LIN {X 0,Y 568.103,Z 672.069,A -85,B 0,C 180,E1 27364.138,E2 27364.138} C_VEL
LIN {X 0,Y 568.021,Z 680.785,A -85,B 0,C 180,E1 27362.825,E2 27362.825} C_VEL
LIN {X 0,Y 567.96,Z 688.715,A -85,B 0,C 180,E1 27361.312,E2 27361.312} C_VEL
LIN {X 0,Y 567.932,Z 694.6,A -85,B 0,C 180,E1 27359.799,E2 27359.799} C_VEL
LIN {X 0,Y 567.918,Z 698.81,A -85,B 0,C 180,E1 27358.285,E2 27358.285} C_VEL
LIN {X 0,Y 567.916,Z 701.625,A -85,B 0,C 180,E1 27356.569,E2 27356.569} C_VEL
LIN {X 0,Y 567.916,Z 702.444,A -85,B 0,C 180,E1 27355.051,E2 27355.051} C_VEL
LIN {X 0,Y 567.916,Z 701.73,A -85,B 0,C 180,E1 27353.429,E2 27353.429} C_VEL
LIN {X 0,Y 567.916,Z 698.96,A -85,B 0,C 180,E1 27351.7,E2 27351.7} C_VEL
LIN {X 0,Y 567.93,Z 694.8,A -85,B 0,C 180,E1 27350.168,E2 27350.168} C_VEL
LIN {X 0,Y 567.961,Z 688.386,A -85,B 0,C 180,E1 27348.526,E2 27348.526} C_VEL
LIN {X 0,Y 568.019,Z 680.765,A -85,B 0,C 180,E1 27347.083,E2 27347.083} C_VEL
LIN {X 0,Y 568.11,Z 671.85,A -85,B 0,C 180,E1 27345.736,E2 27345.736} C_VEL
LIN {X 0,Y 568.235,Z 660.961,A -85,B 0,C 180,E1 27344.435,E2 27344.435} C_VEL
LIN {X 0,Y 568.372,Z 650.225,A -85,B 0,C 180,E1 27343.39,E2 27343.39} C_VEL
LIN {X 0,Y 568.548,Z 637.033,A -85,B 0,C 180,E1 27342.341,E2 27342.341} C_VEL
LIN {X 0,Y 568.727,Z 623.6,A -85,B 0,C 180,E1 27341.502,E2 27341.502} C_VEL
LIN {X 0,Y 568.875,Z 610.751,A -85,B 0,C 180,E1 27340.865,E2 27340.865} C_VEL
LIN {X 0,Y 569.043,Z 595.744,A -85,B 0,C 180,E1 27340.299,E2 27340.299} C_VEL
LIN {X 0,Y 569.158,Z 579.316,A -85,B 0,C 180,E1 27339.884,E2 27339.884} C_VEL
LIN {X 0,Y 569.352,Z 502.923,A -85,B 0,C 180,E1 27338.879,E2 27338.879} C_VEL
LIN {X 0,Y 569.278,Z 438.341,A -85,B 0,C 180,E1 27338.045,E2 27338.045} C_VEL
LIN {X 0,Y 568.987,Z 435.852,A -85,B 0,C 180,E1 27337.992,E2 27337.992} C_VEL
LIN {X 0,Y 569.451,Z 392.592,A -85,B 0,C 180,E1 27334.633,E2 27334.633} C_VEL
LIN {X 0,Y 569.848,Z 350.919,A -85,B 0,C 180,E1 27331.38,E2 27331.38} C_VEL
LIN {X 0,Y 569.783,Z 320.283,A -85,B 0,C 180,E1 27329.105,E2 27329.105} C_VEL
LIN {X 0,Y 569.208,Z 278.696,A -85,B 0,C 180,E1 27326.163,E2 27326.163} C_VEL
LIN {X 0,Y 568.41,Z 243.021,A -85,B 0,C 180,E1 27323.843,E2 27323.843} C_VEL
LIN {X 0,Y 568.206,Z 241.959,A -85,B 0,C 180,E1 27323.755,E2 27323.755} C_VEL
LIN {X 0,Y 568.249,Z 242.205,A -85,B 0,C 180,E1 27322.262,E2 27322.262} C_VEL
LIN {X 0,Y 569.363,Z 245.218,A -85,B 0,C 180,E1 27321.947,E2 27321.947} C_VEL
LIN {X 0,Y 575.363,Z 257.407,A -85,B 0,C 180,E1 27320.568,E2 27320.568} C_VEL
LIN {X 0,Y 574.722,Z 312.789,A -85,B 0,C 180,E1 27316.944,E2 27316.944} C_VEL
LIN {X 0,Y 576.412,Z 325.558,A -85,B 0,C 180,E1 27315.996,E2 27315.996} C_VEL
LIN {X 0,Y 579.316,Z 335.026,A -85,B 0,C 180,E1 27315.183,E2 27315.183} C_VEL
LIN {X 0,Y 583.109,Z 341.733,A -85,B 0,C 180,E1 27314.495,E2 27314.495} C_VEL
LIN {X 0,Y 587.828,Z 346.751,A -85,B 0,C 180,E1 27313.847,E2 27313.847} C_VEL
LIN {X 0,Y 591.052,Z 348.878,A -85,B 0,C 180,E1 27313.33,E2 27313.33} C_VEL
LIN {X 0,Y 593.631,Z 349.586,A -85,B 0,C 180,E1 27312.747,E2 27312.747} C_VEL
LIN {X 0,Y 595.105,Z 348.922,A -85,B 0,C 180,E1 27312.189,E2 27312.189} C_VEL
LIN {X 0,Y 595.528,Z 346.951,A -85,B 0,C 180,E1 27311.608,E2 27311.608} C_VEL
LIN {X 0,Y 594.698,Z 343.734,A -85,B 0,C 180,E1 27311.069,E2 27311.069} C_VEL
LIN {X 0,Y 592.583,Z 339.307,A -85,B 0,C 180,E1 27310.608,E2 27310.608} C_VEL
LIN {X 0,Y 588.547,Z 331.567,A -85,B 0,C 180,E1 27310.129,E2 27310.129} C_VEL
LIN {X 0,Y 585.378,Z 322.433,A -85,B 0,C 180,E1 27309.759,E2 27309.759} C_VEL
LIN {X 0,Y 583.166,Z 311.682,A -85,B 0,C 180,E1 27309.497,E2 27309.497} C_VEL
LIN {X 0,Y 581.969,Z 298.964,A -85,B 0,C 180,E1 27309.355,E2 27309.355} C_VEL
LIN {X 0,Y 581.754,Z 282.03,A -85,B 0,C 180,E1 27309.329,E2 27309.329} C_VEL
LIN {X 0,Y 581.598,Z 258.822,A -85,B 0,C 180,E1 27309.31,E2 27309.31} C_VEL
LIN {X 0,Y 577.973,Z 254.412,A -85,B 0,C 180,E1 27308.869,E2 27308.869} C_VEL
LIN {X 0,Y 574.072,Z 250.389,A -85,B 0,C 180,E1 27308.383,E2 27308.383} C_VEL
LIN {X 0,Y 571.751,Z 250.051,A -85,B 0,C 180,E1 27308.089,E2 27308.089} C_VEL
LIN {X 0,Y 571.629,Z 250.115,A -85,B 0,C 180,E1 27308.043,E2 27308.043} C_VEL
LIN {X 0,Y 573.988,Z 255.905,A -85,B 0,C 180,E1 27307.482,E2 27307.482} C_VEL
LIN {X 0,Y 573.245,Z 302.662,A -85,B 0,C 180,E1 27304.587,E2 27304.587} C_VEL
LIN {X 0,Y 574.384,Z 310.581,A -85,B 0,C 180,E1 27304.391,E2 27304.391} C_VEL
LIN {X 0,Y 573.271,Z 530.669,A -85,B 0,C 180,E1 27301.252,E2 27301.252} C_VEL
LIN {X 0,Y 572.868,Z 608.931,A -85,B 0,C 180,E1 27300.126,E2 27300.126} C_VEL
LIN {X 0,Y 572.55,Z 630.865,A -85,B 0,C 180,E1 27299.618,E2 27299.618} C_VEL
LIN {X 0,Y 572.128,Z 653.445,A -85,B 0,C 180,E1 27298.89,E2 27298.89} C_VEL
LIN {X 0,Y 571.709,Z 674.688,A -85,B 0,C 180,E1 27298.001,E2 27298.001} C_VEL
LIN {X 0,Y 571.187,Z 694.756,A -85,B 0,C 180,E1 27296.961,E2 27296.961} C_VEL
LIN {X 0,Y 570.674,Z 714.156,A -85,B 0,C 180,E1 27295.754,E2 27295.754} C_VEL
LIN {X 0,Y 570.184,Z 732.799,A -85,B 0,C 180,E1 27294.391,E2 27294.391} C_VEL
LIN {X 0,Y 569.662,Z 751.692,A -85,B 0,C 180,E1 27292.769,E2 27292.769} C_VEL
LIN {X 0,Y 569.196,Z 769.23,A -85,B 0,C 180,E1 27290.999,E2 27290.999} C_VEL
LIN {X 0,Y 568.818,Z 784.581,A -85,B 0,C 180,E1 27289.19,E2 27289.19} C_VEL
LIN {X 0,Y 568.521,Z 798.676,A -85,B 0,C 180,E1 27287.259,E2 27287.259} C_VEL
LIN {X 0,Y 568.303,Z 810.938,A -85,B 0,C 180,E1 27285.302,E2 27285.302} C_VEL
LIN {X 0,Y 568.132,Z 821.9,A -85,B 0,C 180,E1 27283.226,E2 27283.226} C_VEL
LIN {X 0,Y 568.021,Z 830.897,A -85,B 0,C 180,E1 27281.165,E2 27281.165} C_VEL
LIN {X 0,Y 567.965,Z 838.562,A -85,B 0,C 180,E1 27279.014,E2 27279.014} C_VEL
LIN {X 0,Y 567.933,Z 844.578,A -85,B 0,C 180,E1 27276.817,E2 27276.817} C_VEL
LIN {X 0,Y 567.916,Z 848.793,A -85,B 0,C 180,E1 27274.645,E2 27274.645} C_VEL
LIN {X 0,Y 567.909,Z 851.489,A -85,B 0,C 180,E1 27272.422,E2 27272.422} C_VEL
LIN {X 0,Y 567.905,Z 852.475,A -85,B 0,C 180,E1 27270.202,E2 27270.202} C_VEL
LIN {X 0,Y 567.912,Z 851.758,A -85,B 0,C 180,E1 27267.982,E2 27267.982} C_VEL
LIN {X 0,Y 567.914,Z 849.426,A -85,B 0,C 180,E1 27265.759,E2 27265.759} C_VEL
LIN {X 0,Y 567.915,Z 845.586,A -85,B 0,C 180,E1 27263.632,E2 27263.632} C_VEL
LIN {X 0,Y 567.937,Z 840.08,A -85,B 0,C 180,E1 27261.496,E2 27261.496} C_VEL
LIN {X 0,Y 567.996,Z 833.316,A -85,B 0,C 180,E1 27259.451,E2 27259.451} C_VEL
LIN {X 0,Y 568.086,Z 824.764,A -85,B 0,C 180,E1 27257.394,E2 27257.394} C_VEL
LIN {X 0,Y 568.235,Z 813.833,A -85,B 0,C 180,E1 27255.218,E2 27255.218} C_VEL
LIN {X 0,Y 568.458,Z 801.998,A -85,B 0,C 180,E1 27253.234,E2 27253.234} C_VEL
LIN {X 0,Y 568.759,Z 787.904,A -85,B 0,C 180,E1 27251.234,E2 27251.234} C_VEL
LIN {X 0,Y 569.106,Z 773.042,A -85,B 0,C 180,E1 27249.428,E2 27249.428} C_VEL
LIN {X 0,Y 569.526,Z 756.535,A -85,B 0,C 180,E1 27247.698,E2 27247.698} C_VEL
LIN {X 0,Y 569.994,Z 738.779,A -85,B 0,C 180,E1 27246.095,E2 27246.095} C_VEL
LIN {X 0,Y 570.521,Z 720.526,A -85,B 0,C 180,E1 27244.683,E2 27244.683} C_VEL
LIN {X 0,Y 571.06,Z 700.433,A -85,B 0,C 180,E1 27243.37,E2 27243.37} C_VEL
LIN {X 0,Y 571.525,Z 680.177,A -85,B 0,C 180,E1 27242.266,E2 27242.266} C_VEL
LIN {X 0,Y 572.038,Z 659.333,A -85,B 0,C 180,E1 27241.335,E2 27241.335} C_VEL
LIN {X 0,Y 572.456,Z 637.558,A -85,B 0,C 180,E1 27240.574,E2 27240.574} C_VEL
LIN {X 0,Y 572.759,Z 615.949,A -85,B 0,C 180,E1 27240.017,E2 27240.017} C_VEL
LIN {X 0,Y 573.002,Z 591.483,A -85,B 0,C 180,E1 27239.601,E2 27239.601} C_VEL
LIN {X 0,Y 574.056,Z 367.034,A -85,B 0,C 180,E1 27236.421,E2 27236.421} C_VEL
LIN {X 0,Y 574.187,Z 309.846,A -85,B 0,C 180,E1 27235.584,E2 27235.584} C_VEL
LIN {X 0,Y 572.736,Z 302.398,A -85,B 0,C 180,E1 27235.347,E2 27235.347} C_VEL
LIN {X 0,Y 573.538,Z 262.173,A -85,B 0,C 180,E1 27232.398,E2 27232.398} C_VEL
LIN {X 0,Y 573.705,Z 255.551,A -85,B 0,C 180,E1 27231.905,E2 27231.905} C_VEL
LIN {X 0,Y 573.143,Z 254.07,A -85,B 0,C 180,E1 27231.734,E2 27231.734} C_VEL
LIN {X 0,Y 575.005,Z 254.784,A -85,B 0,C 180,E1 27231.5,E2 27231.5} C_VEL
LIN {X 0,Y 577.504,Z 253.868,A -85,B 0,C 180,E1 27231.189,E2 27231.189} C_VEL
LIN {X 0,Y 581.598,Z 258.84,A -85,B 0,C 180,E1 27230.69,E2 27230.69} C_VEL
LIN {X 0,Y 581.762,Z 267.678,A -85,B 0,C 180,E1 27230.67,E2 27230.67} C_VEL
LIN {X 0,Y 581.94,Z 336.852,A -85,B 0,C 180,E1 27230.649,E2 27230.649} C_VEL
LIN {X 0,Y 583.106,Z 349.267,A -85,B 0,C 180,E1 27230.51,E2 27230.51} C_VEL
LIN {X 0,Y 585.298,Z 359.813,A -85,B 0,C 180,E1 27230.25,E2 27230.25} C_VEL
LIN {X 0,Y 588.468,Z 368.899,A -85,B 0,C 180,E1 27229.88,E2 27229.88} C_VEL
LIN {X 0,Y 591.818,Z 375.728,A -85,B 0,C 180,E1 27229.456,E2 27229.456} C_VEL
LIN {X 0,Y 593.551,Z 380.22,A -85,B 0,C 180,E1 27228.985,E2 27228.985} C_VEL
LIN {X 0,Y 594.01,Z 383.359,A -85,B 0,C 180,E1 27228.456,E2 27228.456} C_VEL
LIN {X 0,Y 593.268,Z 385.325,A -85,B 0,C 180,E1 27227.863,E2 27227.863} C_VEL
LIN {X 0,Y 591.619,Z 385.905,A -85,B 0,C 180,E1 27227.321,E2 27227.321} C_VEL
LIN {X 0,Y 588.94,Z 385.128,A -85,B 0,C 180,E1 27226.746,E2 27226.746} C_VEL
LIN {X 0,Y 585.706,Z 382.882,A -85,B 0,C 180,E1 27226.228,E2 27226.228} C_VEL
LIN {X 0,Y 580.98,Z 377.491,A -85,B 0,C 180,E1 27225.537,E2 27225.537} C_VEL
LIN {X 0,Y 577.144,Z 369.886,A -85,B 0,C 180,E1 27224.741,E2 27224.741} C_VEL
LIN {X 0,Y 574.585,Z 359.77,A -85,B 0,C 180,E1 27223.834,E2 27223.834} C_VEL
LIN {X 0,Y 573.474,Z 347.302,A -85,B 0,C 180,E1 27222.841,E2 27222.841} C_VEL
LIN {X 0,Y 574.378,Z 298.185,A -85,B 0,C 180,E1 27219.19,E2 27219.19} C_VEL
LIN {X 0,Y 575.319,Z 262.814,A -85,B 0,C 180,E1 27216.422,E2 27216.422} C_VEL
LIN {X 0,Y 575.444,Z 257.912,A -85,B 0,C 180,E1 27216.026,E2 27216.026} C_VEL
LIN {X 0,Y 569.719,Z 245.758,A -85,B 0,C 180,E1 27214.41,E2 27214.41} C_VEL
LIN {X 0,Y 568.261,Z 242.304,A -85,B 0,C 180,E1 27213.952,E2 27213.952} C_VEL
LIN {X 0,Y 568.218,Z 241.96,A -85,B 0,C 180,E1 27213.844,E2 27213.844} C_VEL
LIN {X 0,Y 568.212,Z 241.956,A -85,B 0,C 180,E1 27210.566,E2 27210.566} C_VEL
LIN {X 0,Y 568.193,Z 241.957,A -85,B 0,C 180,E1 27207.294,E2 27207.294} C_VEL
LIN {X 0,Y 568.248,Z 242.138,A -85,B 0,C 180,E1 27206.772,E2 27206.772} C_VEL
LIN {X 0,Y 568.786,Z 246.032,A -85,B 0,C 180,E1 27206.519,E2 27206.519} C_VEL
LIN {X 0,Y 569.334,Z 290.314,A -85,B 0,C 180,E1 27203.713,E2 27203.713} C_VEL
LIN {X 0,Y 569.709,Z 330.255,A -85,B 0,C 180,E1 27201.027,E2 27201.027} C_VEL
LIN {X 0,Y 569.686,Z 369.499,A -85,B 0,C 180,E1 27198.283,E2 27198.283} C_VEL
LIN {X 0,Y 569.314,Z 415.814,A -85,B 0,C 180,E1 27194.961,E2 27194.961} C_VEL
LIN {X 0,Y 568.878,Z 462.441,A -85,B 0,C 180,E1 27191.609,E2 27191.609} C_VEL
LIN {X 0,Y 568.719,Z 486.046,A -85,B 0,C 180,E1 27189.958,E2 27189.958} C_VEL
LIN {X 0,Y 568.974,Z 504.828,A -85,B 0,C 180,E1 27189.712,E2 27189.712} C_VEL
LIN {X 0,Y 568.782,Z 600.137,A -85,B 0,C 180,E1 27188.478,E2 27188.478} C_VEL
LIN {X 0,Y 568.673,Z 614.305,A -85,B 0,C 180,E1 27188.113,E2 27188.113} C_VEL
LIN {X 0,Y 568.546,Z 629.275,A -85,B 0,C 180,E1 27187.528,E2 27187.528} C_VEL
LIN {X 0,Y 568.411,Z 641.437,A -85,B 0,C 180,E1 27186.87,E2 27186.87} C_VEL
LIN {X 0,Y 568.292,Z 653.855,A -85,B 0,C 180,E1 27186.009,E2 27186.009} C_VEL
LIN {X 0,Y 568.171,Z 664.604,A -85,B 0,C 180,E1 27185.048,E2 27185.048} C_VEL
LIN {X 0,Y 568.077,Z 673.742,A -85,B 0,C 180,E1 27184.037,E2 27184.037} C_VEL
LIN {X 0,Y 568.005,Z 682.503,A -85,B 0,C 180,E1 27182.825,E2 27182.825} C_VEL
LIN {X 0,Y 567.956,Z 689.743,A -85,B 0,C 180,E1 27181.513,E2 27181.513} C_VEL
LIN {X 0,Y 567.932,Z 695.583,A -85,B 0,C 180,E1 27180.101,E2 27180.101} C_VEL
LIN {X 0,Y 567.918,Z 699.492,A -85,B 0,C 180,E1 27178.688,E2 27178.688} C_VEL
LIN {X 0,Y 567.918,Z 701.784,A -85,B 0,C 180,E1 27177.275,E2 27177.275} C_VEL
LIN {X 0,Y 567.916,Z 702.435,A -85,B 0,C 180,E1 27175.658,E2 27175.658} C_VEL
LIN {X 0,Y 567.915,Z 701.297,A -85,B 0,C 180,E1 27174.24,E2 27174.24} C_VEL
LIN {X 0,Y 567.922,Z 698.323,A -85,B 0,C 180,E1 27172.717,E2 27172.717} C_VEL
LIN {X 0,Y 567.937,Z 693.636,A -85,B 0,C 180,E1 27171.291,E2 27171.291} C_VEL
LIN {X 0,Y 567.969,Z 687.598,A -85,B 0,C 180,E1 27169.963,E2 27169.963} C_VEL
LIN {X 0,Y 568.026,Z 679.425,A -85,B 0,C 180,E1 27168.629,E2 27168.629} C_VEL
LIN {X 0,Y 568.111,Z 670.597,A -85,B 0,C 180,E1 27167.497,E2 27167.497} C_VEL
LIN {X 0,Y 568.231,Z 659.29,A -85,B 0,C 180,E1 27166.362,E2 27166.362} C_VEL
LIN {X 0,Y 568.334,Z 648.145,A -85,B 0,C 180,E1 27165.481,E2 27165.481} C_VEL
LIN {X 0,Y 568.491,Z 635.69,A -85,B 0,C 180,E1 27164.703,E2 27164.703} C_VEL
LIN {X 0,Y 568.594,Z 622.162,A -85,B 0,C 180,E1 27164.078,E2 27164.078} C_VEL
LIN {X 0,Y 568.685,Z 611.706,A -85,B 0,C 180,E1 27163.718,E2 27163.718} C_VEL
LIN {X 0,Y 568.08,Z 605.34,A -85,B 0,C 180,E1 27163.528,E2 27163.528} C_VEL
LIN {X 0,Y 564.229,Z 592.883,A -85,B 0,C 180,E1 27163.207,E2 27163.207} C_VEL
LIN {X 0,Y 561.555,Z 583.373,A -85,B 0,C 180,E1 27163.022,E2 27163.022} C_VEL
LIN {X 0,Y 561.029,Z 577.907,A -85,B 0,C 180,E1 27162.942,E2 27162.942} C_VEL
LIN {X 0,Y 560.996,Z 487.134,A -85,B 0,C 180,E1 27161.77,E2 27161.77} C_VEL
LIN {X 0,Y 560.849,Z 485.137,A -85,B 0,C 180,E1 27161.713,E2 27161.713} C_VEL
LIN {X 0,Y 561.334,Z 440.472,A -85,B 0,C 180,E1 27158.473,E2 27158.473} C_VEL
LIN {X 0,Y 561.732,Z 406.576,A -85,B 0,C 180,E1 27156.001,E2 27156.001} C_VEL
LIN {X 0,Y 562.152,Z 365.369,A -85,B 0,C 180,E1 27153.012,E2 27153.012} C_VEL
LIN {X 0,Y 562.413,Z 332.203,A -85,B 0,C 180,E1 27150.59,E2 27150.59} C_VEL
LIN {X 0,Y 562.503,Z 289.911,A -85,B 0,C 180,E1 27147.533,E2 27147.533} C_VEL
LIN {X 0,Y 562.54,Z 250.875,A -85,B 0,C 180,E1 27144.714,E2 27144.714} C_VEL
LIN {X 0,Y 560.284,Z 242.946,A -85,B 0,C 180,E1 27144.015,E2 27144.015} C_VEL
LIN {X 0,Y 560.244,Z 242.949,A -85,B 0,C 180,E1 27140.686,E2 27140.686} C_VEL
LIN {X 0,Y 560.282,Z 242.948,A -85,B 0,C 180,E1 27137.301,E2 27137.301} C_VEL
LIN {X 0,Y 560.284,Z 242.946,A -85,B 0,C 180,E1 27133.822,E2 27133.822} C_VEL
LIN {X 0,Y 560.249,Z 242.95,A -85,B 0,C 180,E1 27130.511,E2 27130.511} C_VEL
LIN {X 0,Y 560.307,Z 243.182,A -85,B 0,C 180,E1 27128.854,E2 27128.854} C_VEL
LIN {X 0,Y 561.827,Z 246.79,A -85,B 0,C 180,E1 27128.294,E2 27128.294} C_VEL
LIN {X 0,Y 564.705,Z 256.207,A -85,B 0,C 180,E1 27126.957,E2 27126.957} C_VEL
LIN {X 0,Y 563.871,Z 291.566,A -85,B 0,C 180,E1 27123.773,E2 27123.773} C_VEL
LIN {X 0,Y 563.805,Z 300.759,A -85,B 0,C 180,E1 27122.99,E2 27122.99} C_VEL
LIN {X 0,Y 565.652,Z 310.153,A -85,B 0,C 180,E1 27122.747,E2 27122.747} C_VEL
LIN {X 0,Y 564.54,Z 542.616,A -85,B 0,C 180,E1 27119.524,E2 27119.524} C_VEL
LIN {X 0,Y 564.313,Z 566.976,A -85,B 0,C 180,E1 27119.122,E2 27119.122} C_VEL
LIN {X 0,Y 563.97,Z 587.827,A -85,B 0,C 180,E1 27118.582,E2 27118.582} C_VEL
LIN {X 0,Y 563.618,Z 606.295,A -85,B 0,C 180,E1 27117.927,E2 27117.927} C_VEL
LIN {X 0,Y 563.163,Z 626.085,A -85,B 0,C 180,E1 27117.034,E2 27117.034} C_VEL
LIN {X 0,Y 562.677,Z 643.798,A -85,B 0,C 180,E1 27116.035,E2 27116.035} C_VEL
LIN {X 0,Y 562.188,Z 661.902,A -85,B 0,C 180,E1 27114.818,E2 27114.818} C_VEL
LIN {X 0,Y 561.692,Z 678.921,A -85,B 0,C 180,E1 27113.444,E2 27113.444} C_VEL
LIN {X 0,Y 561.262,Z 694.552,A -85,B 0,C 180,E1 27111.969,E2 27111.969} C_VEL
LIN {X 0,Y 560.841,Z 710.006,A -85,B 0,C 180,E1 27110.235,E2 27110.235} C_VEL
LIN {X 0,Y 560.544,Z 723.083,A -85,B 0,C 180,E1 27108.512,E2 27108.512} C_VEL
LIN {X 0,Y 560.294,Z 735.336,A -85,B 0,C 180,E1 27106.59,E2 27106.59} C_VEL
LIN {X 0,Y 560.119,Z 744.904,A -85,B 0,C 180,E1 27104.79,E2 27104.79} C_VEL
LIN {X 0,Y 560.011,Z 753.713,A -85,B 0,C 180,E1 27102.791,E2 27102.791} C_VEL
LIN {X 0,Y 559.953,Z 760.638,A -85,B 0,C 180,E1 27100.806,E2 27100.806} C_VEL
LIN {X 0,Y 559.928,Z 766.157,A -85,B 0,C 180,E1 27098.73,E2 27098.73} C_VEL
LIN {X 0,Y 559.912,Z 770.011,A -85,B 0,C 180,E1 27096.563,E2 27096.563} C_VEL
LIN {X 0,Y 559.906,Z 771.999,A -85,B 0,C 180,E1 27094.507,E2 27094.507} C_VEL
LIN {X 0,Y 559.902,Z 772.39,A -85,B 0,C 180,E1 27092.354,E2 27092.354} C_VEL
LIN {X 0,Y 559.911,Z 771.03,A -85,B 0,C 180,E1 27090.205,E2 27090.205} C_VEL
LIN {X 0,Y 559.922,Z 767.914,A -85,B 0,C 180,E1 27088.056,E2 27088.056} C_VEL
LIN {X 0,Y 559.944,Z 763.246,A -85,B 0,C 180,E1 27086.007,E2 27086.007} C_VEL
LIN {X 0,Y 559.993,Z 756.846,A -85,B 0,C 180,E1 27083.953,E2 27083.953} C_VEL
LIN {X 0,Y 560.077,Z 748.537,A -85,B 0,C 180,E1 27081.892,E2 27081.892} C_VEL
LIN {X 0,Y 560.227,Z 738.758,A -85,B 0,C 180,E1 27079.927,E2 27079.927} C_VEL
LIN {X 0,Y 560.441,Z 727.488,A -85,B 0,C 180,E1 27078.056,E2 27078.056} C_VEL
LIN {X 0,Y 560.729,Z 714.878,A -85,B 0,C 180,E1 27076.281,E2 27076.281} C_VEL
LIN {X 0,Y 561.107,Z 699.767,A -85,B 0,C 180,E1 27074.497,E2 27074.497} C_VEL
LIN {X 0,Y 561.512,Z 685.107,A -85,B 0,C 180,E1 27073.021,E2 27073.021} C_VEL
LIN {X 0,Y 562.012,Z 667.773,A -85,B 0,C 180,E1 27071.538,E2 27071.538} C_VEL
LIN {X 0,Y 562.47,Z 651.501,A -85,B 0,C 180,E1 27070.368,E2 27070.368} C_VEL
LIN {X 0,Y 562.97,Z 633.082,A -85,B 0,C 180,E1 27069.248,E2 27069.248} C_VEL
LIN {X 0,Y 563.414,Z 614.666,A -85,B 0,C 180,E1 27068.338,E2 27068.338} C_VEL
LIN {X 0,Y 563.824,Z 596.494,A -85,B 0,C 180,E1 27067.615,E2 27067.615} C_VEL
LIN {X 0,Y 564.194,Z 575.342,A -85,B 0,C 180,E1 27066.977,E2 27066.977} C_VEL
LIN {X 0,Y 564.442,Z 555.321,A -85,B 0,C 180,E1 27066.572,E2 27066.572} C_VEL
LIN {X 0,Y 565.67,Z 312.922,A -85,B 0,C 180,E1 27063.204,E2 27063.204} C_VEL
LIN {X 0,Y 565.434,Z 306.062,A -85,B 0,C 180,E1 27063.092,E2 27063.092} C_VEL
LIN {X 0,Y 564.126,Z 299.083,A -85,B 0,C 180,E1 27062.902,E2 27062.902} C_VEL
LIN {X 0,Y 565.041,Z 256.12,A -85,B 0,C 180,E1 27059.626,E2 27059.626} C_VEL
LIN {X 0,Y 561.938,Z 247.476,A -85,B 0,C 180,E1 27058.658,E2 27058.658} C_VEL
LIN {X 0,Y 560.275,Z 242.948,A -85,B 0,C 180,E1 27058.053,E2 27058.053} C_VEL
LIN {X 0,Y 560.269,Z 242.95,A -85,B 0,C 180,E1 27054.8,E2 27054.8} C_VEL
LIN {X 0,Y 560.265,Z 242.951,A -85,B 0,C 180,E1 27051.476,E2 27051.476} C_VEL
LIN {X 0,Y 560.275,Z 242.949,A -85,B 0,C 180,E1 27048.089,E2 27048.089} C_VEL
LIN {X 0,Y 560.273,Z 242.947,A -85,B 0,C 180,E1 27044.743,E2 27044.743} C_VEL
LIN {X 0,Y 560.266,Z 242.946,A -85,B 0,C 180,E1 27041.324,E2 27041.324} C_VEL
LIN {X 0,Y 560.282,Z 242.944,A -85,B 0,C 180,E1 27038.001,E2 27038.001} C_VEL
LIN {X 0,Y 560.265,Z 242.948,A -85,B 0,C 180,E1 27034.643,E2 27034.643} C_VEL
LIN {X 0,Y 560.268,Z 242.948,A -85,B 0,C 180,E1 27031.287,E2 27031.287} C_VEL
LIN {X 0,Y 560.277,Z 242.948,A -85,B 0,C 180,E1 27027.876,E2 27027.876} C_VEL
LIN {X 0,Y 560.261,Z 242.977,A -85,B 0,C 180,E1 27027.453,E2 27027.453} C_VEL
LIN {X 0,Y 562.74,Z 252.348,A -85,B 0,C 180,E1 27026.6,E2 27026.6} C_VEL
LIN {X 0,Y 562.669,Z 297.517,A -85,B 0,C 180,E1 27023.066,E2 27023.066} C_VEL
LIN {X 0,Y 562.435,Z 336.396,A -85,B 0,C 180,E1 27020.012,E2 27020.012} C_VEL
LIN {X 0,Y 562.023,Z 376.635,A -85,B 0,C 180,E1 27016.838,E2 27016.838} C_VEL
LIN {X 0,Y 561.494,Z 413.572,A -85,B 0,C 180,E1 27013.91,E2 27013.91} C_VEL
LIN {X 0,Y 561.272,Z 436.474,A -85,B 0,C 180,E1 27012.138,E2 27012.138} C_VEL
LIN {X 0,Y 561.824,Z 444.029,A -85,B 0,C 180,E1 27012.022,E2 27012.022} C_VEL
LIN {X 0,Y 561.425,Z 577.922,A -85,B 0,C 180,E1 27010.259,E2 27010.259} C_VEL
LIN {X 0,Y 561.302,Z 594.042,A -85,B 0,C 180,E1 27009.873,E2 27009.873} C_VEL
LIN {X 0,Y 561.118,Z 608.695,A -85,B 0,C 180,E1 27009.332,E2 27009.332} C_VEL
LIN {X 0,Y 560.928,Z 621.48,A -85,B 0,C 180,E1 27008.715,E2 27008.715} C_VEL
LIN {X 0,Y 560.713,Z 635.736,A -85,B 0,C 180,E1 27007.841,E2 27007.841} C_VEL
LIN {X 0,Y 560.501,Z 648.758,A -85,B 0,C 180,E1 27006.813,E2 27006.813} C_VEL
LIN {X 0,Y 560.336,Z 658.941,A -85,B 0,C 180,E1 27005.838,E2 27005.838} C_VEL
LIN {X 0,Y 560.188,Z 669.591,A -85,B 0,C 180,E1 27004.607,E2 27004.607} C_VEL
LIN {X 0,Y 560.056,Z 679.365,A -85,B 0,C 180,E1 27003.173,E2 27003.173} C_VEL
LIN {X 0,Y 559.985,Z 686.62,A -85,B 0,C 180,E1 27001.842,E2 27001.842} C_VEL
LIN {X 0,Y 559.945,Z 693.135,A -85,B 0,C 180,E1 27000.307,E2 27000.307} C_VEL
LIN {X 0,Y 559.921,Z 697.743,A -85,B 0,C 180,E1 26998.773,E2 26998.773} C_VEL
LIN {X 0,Y 559.917,Z 700.79,A -85,B 0,C 180,E1 26997.237,E2 26997.237} C_VEL
LIN {X 0,Y 559.914,Z 702.385,A -85,B 0,C 180,E1 26995.494,E2 26995.494} C_VEL
LIN {X 0,Y 559.916,Z 702.114,A -85,B 0,C 180,E1 26993.953,E2 26993.953} C_VEL
LIN {X 0,Y 559.92,Z 700.381,A -85,B 0,C 180,E1 26992.407,E2 26992.407} C_VEL
LIN {X 0,Y 559.927,Z 696.472,A -85,B 0,C 180,E1 26990.648,E2 26990.648} C_VEL
LIN {X 0,Y 559.951,Z 691.328,A -85,B 0,C 180,E1 26989.142,E2 26989.142} C_VEL
LIN {X 0,Y 560.009,Z 684.465,A -85,B 0,C 180,E1 26987.629,E2 26987.629} C_VEL
LIN {X 0,Y 560.101,Z 675.686,A -85,B 0,C 180,E1 26986.161,E2 26986.161} C_VEL
LIN {X 0,Y 560.226,Z 666.441,A -85,B 0,C 180,E1 26984.918,E2 26984.918} C_VEL
LIN {X 0,Y 560.399,Z 655.577,A -85,B 0,C 180,E1 26983.72,E2 26983.72} C_VEL
LIN {X 0,Y 560.584,Z 643.693,A -85,B 0,C 180,E1 26982.671,E2 26982.671} C_VEL
LIN {X 0,Y 560.762,Z 631.902,A -85,B 0,C 180,E1 26981.819,E2 26981.819} C_VEL
LIN {X 0,Y 560.991,Z 618.241,A -85,B 0,C 180,E1 26981.018,E2 26981.018} C_VEL
LIN {X 0,Y 561.208,Z 602.372,A -85,B 0,C 180,E1 26980.323,E2 26980.323} C_VEL
LIN {X 0,Y 561.37,Z 586.423,A -85,B 0,C 180,E1 26979.829,E2 26979.829} C_VEL
LIN {X 0,Y 561.486,Z 569.992,A -85,B 0,C 180,E1 26979.522,E2 26979.522} C_VEL
LIN {X 0,Y 561.622,Z 439.155,A -85,B 0,C 180,E1 26977.818,E2 26977.818} C_VEL
LIN {X 0,Y 561.229,Z 435.788,A -85,B 0,C 180,E1 26977.746,E2 26977.746} C_VEL
LIN {X 0,Y 561.844,Z 394.425,A -85,B 0,C 180,E1 26974.457,E2 26974.457} C_VEL
LIN {X 0,Y 562.133,Z 351.099,A -85,B 0,C 180,E1 26971.125,E2 26971.125} C_VEL
LIN {X 0,Y 562.03,Z 319.103,A -85,B 0,C 180,E1 26968.767,E2 26968.767} C_VEL
LIN {X 0,Y 561.642,Z 292.203,A -85,B 0,C 180,E1 26966.871,E2 26966.871} C_VEL
LIN {X 0,Y 560.94,Z 262.205,A -85,B 0,C 180,E1 26964.849,E2 26964.849} C_VEL
LIN {X 0,Y 560.562,Z 244.404,A -85,B 0,C 180,E1 26963.729,E2 26963.729} C_VEL
LIN {X 0,Y 560.272,Z 242.948,A -85,B 0,C 180,E1 26963.632,E2 26963.632} C_VEL
LIN {X 0,Y 560.318,Z 243.188,A -85,B 0,C 180,E1 26962.943,E2 26962.943} C_VEL
LIN {X 0,Y 561.481,Z 246.266,A -85,B 0,C 180,E1 26962.61,E2 26962.61} C_VEL
LIN {X 0,Y 568.076,Z 259.489,A -85,B 0,C 180,E1 26961.072,E2 26961.072} C_VEL
LIN {X 0,Y 568.856,Z 261.317,A -85,B 0,C 180,E1 26960.876,E2 26960.876} C_VEL
LIN {X 0,Y 568.016,Z 314.894,A -85,B 0,C 180,E1 26957.336,E2 26957.336} C_VEL
LIN {X 0,Y 569.532,Z 327.807,A -85,B 0,C 180,E1 26956.375,E2 26956.375} C_VEL
LIN {X 0,Y 572.482,Z 338.361,A -85,B 0,C 180,E1 26955.474,E2 26955.474} C_VEL
LIN {X 0,Y 576.569,Z 346.167,A -85,B 0,C 180,E1 26954.684,E2 26954.684} C_VEL
LIN {X 0,Y 581.839,Z 352.146,A -85,B 0,C 180,E1 26953.944,E2 26953.944} C_VEL
LIN {X 0,Y 586.219,Z 355.343,A -85,B 0,C 180,E1 26953.399,E2 26953.399} C_VEL
LIN {X 0,Y 589.456,Z 356.694,A -85,B 0,C 180,E1 26952.859,E2 26952.859} C_VEL
LIN {X 0,Y 591.855,Z 356.661,A -85,B 0,C 180,E1 26952.25,E2 26952.25} C_VEL
LIN {X 0,Y 593.025,Z 355.201,A -85,B 0,C 180,E1 26951.629,E2 26951.629} C_VEL
LIN {X 0,Y 592.812,Z 352.498,A -85,B 0,C 180,E1 26951.041,E2 26951.041} C_VEL
LIN {X 0,Y 591.242,Z 348.756,A -85,B 0,C 180,E1 26950.528,E2 26950.528} C_VEL
LIN {X 0,Y 588.225,Z 343.709,A -85,B 0,C 180,E1 26950.092,E2 26950.092} C_VEL
LIN {X 0,Y 583.98,Z 335.296,A -85,B 0,C 180,E1 26949.595,E2 26949.595} C_VEL
LIN {X 0,Y 580.649,Z 325.388,A -85,B 0,C 180,E1 26949.195,E2 26949.195} C_VEL
LIN {X 0,Y 578.326,Z 314.083,A -85,B 0,C 180,E1 26948.912,E2 26948.912} C_VEL
LIN {X 0,Y 577.013,Z 300.916,A -85,B 0,C 180,E1 26948.751,E2 26948.751} C_VEL
LIN {X 0,Y 576.718,Z 284.457,A -85,B 0,C 180,E1 26948.714,E2 26948.714} C_VEL
LIN {X 0,Y 576.564,Z 263.083,A -85,B 0,C 180,E1 26948.695,E2 26948.695} C_VEL
LIN {X 0,Y 574.072,Z 260.1,A -85,B 0,C 180,E1 26948.383,E2 26948.383} C_VEL
LIN {X 0,Y 572.987,Z 259.361,A -85,B 0,C 180,E1 26948.246,E2 26948.246} C_VEL
LIN {X 0,Y 568.987,Z 263.829,A -85,B 0,C 180,E1 26947.732,E2 26947.732} C_VEL
LIN {X 0,Y 567.308,Z 264.07,A -85,B 0,C 180,E1 26947.513,E2 26947.513} C_VEL
LIN {X 0,Y 567.112,Z 264.046,A -85,B 0,C 180,E1 26947.48,E2 26947.48} C_VEL
LIN {X 0,Y 566.396,Z 302.665,A -85,B 0,C 180,E1 26945.066,E2 26945.066} C_VEL
LIN {X 0,Y 567.773,Z 311.977,A -85,B 0,C 180,E1 26944.828,E2 26944.828} C_VEL
LIN {X 0,Y 566.424,Z 531.814,A -85,B 0,C 180,E1 26941.656,E2 26941.656} C_VEL
LIN {X 0,Y 565.943,Z 608.918,A -85,B 0,C 180,E1 26940.534,E2 26940.534} C_VEL
LIN {X 0,Y 565.556,Z 631.023,A -85,B 0,C 180,E1 26940.018,E2 26940.018} C_VEL
LIN {X 0,Y 565.047,Z 654.002,A -85,B 0,C 180,E1 26939.265,E2 26939.265} C_VEL
LIN {X 0,Y 564.547,Z 674.568,A -85,B 0,C 180,E1 26938.394,E2 26938.394} C_VEL
LIN {X 0,Y 563.915,Z 694.763,A -85,B 0,C 180,E1 26937.337,E2 26937.337} C_VEL
LIN {X 0,Y 563.284,Z 714.677,A -85,B 0,C 180,E1 26936.081,E2 26936.081} C_VEL
LIN {X 0,Y 562.65,Z 734.153,A -85,B 0,C 180,E1 26934.628,E2 26934.628} C_VEL
LIN {X 0,Y 562.043,Z 752.269,A -85,B 0,C 180,E1 26933.04,E2 26933.04} C_VEL
LIN {X 0,Y 561.48,Z 769.731,A -85,B 0,C 180,E1 26931.247,E2 26931.247} C_VEL
LIN {X 0,Y 561.013,Z 785.432,A -85,B 0,C 180,E1 26929.36,E2 26929.36} C_VEL
LIN {X 0,Y 560.656,Z 799.224,A -85,B 0,C 180,E1 26927.427,E2 26927.427} C_VEL
LIN {X 0,Y 560.383,Z 811.522,A -85,B 0,C 180,E1 26925.418,E2 26925.418} C_VEL
LIN {X 0,Y 560.18,Z 822.404,A -85,B 0,C 180,E1 26923.312,E2 26923.312} C_VEL
LIN {X 0,Y 560.045,Z 831.308,A -85,B 0,C 180,E1 26921.221,E2 26921.221} C_VEL
LIN {X 0,Y 559.964,Z 839.172,A -85,B 0,C 180,E1 26918.937,E2 26918.937} C_VEL
LIN {X 0,Y 559.935,Z 844.923,A -85,B 0,C 180,E1 26916.768,E2 26916.768} C_VEL
LIN {X 0,Y 559.917,Z 848.954,A -85,B 0,C 180,E1 26914.609,E2 26914.609} C_VEL
LIN {X 0,Y 559.91,Z 851.559,A -85,B 0,C 180,E1 26912.354,E2 26912.354} C_VEL
LIN {X 0,Y 559.911,Z 852.489,A -85,B 0,C 180,E1 26910.102,E2 26910.102} C_VEL
LIN {X 0,Y 559.912,Z 851.693,A -85,B 0,C 180,E1 26907.851,E2 26907.851} C_VEL
LIN {X 0,Y 559.916,Z 849.271,A -85,B 0,C 180,E1 26905.596,E2 26905.596} C_VEL
LIN {X 0,Y 559.921,Z 845.377,A -85,B 0,C 180,E1 26903.437,E2 26903.437} C_VEL
LIN {X 0,Y 559.949,Z 839.78,A -85,B 0,C 180,E1 26901.27,E2 26901.27} C_VEL
LIN {X 0,Y 560.024,Z 832.531,A -85,B 0,C 180,E1 26899.091,E2 26899.091} C_VEL
LIN {X 0,Y 560.155,Z 823.379,A -85,B 0,C 180,E1 26896.898,E2 26896.898} C_VEL
LIN {X 0,Y 560.348,Z 812.679,A -85,B 0,C 180,E1 26894.793,E2 26894.793} C_VEL
LIN {X 0,Y 560.637,Z 799.882,A -85,B 0,C 180,E1 26892.672,E2 26892.672} C_VEL
LIN {X 0,Y 560.995,Z 786.279,A -85,B 0,C 180,E1 26890.748,E2 26890.748} C_VEL
LIN {X 0,Y 561.468,Z 770.221,A -85,B 0,C 180,E1 26888.807,E2 26888.807} C_VEL
LIN {X 0,Y 562.023,Z 752.828,A -85,B 0,C 180,E1 26887.014,E2 26887.014} C_VEL
LIN {X 0,Y 562.627,Z 734.817,A -85,B 0,C 180,E1 26885.427,E2 26885.427} C_VEL
LIN {X 0,Y 563.244,Z 715.764,A -85,B 0,C 180,E1 26883.993,E2 26883.993} C_VEL
LIN {X 0,Y 563.892,Z 695.755,A -85,B 0,C 180,E1 26882.719,E2 26882.719} C_VEL
LIN {X 0,Y 564.508,Z 675.708,A -85,B 0,C 180,E1 26881.661,E2 26881.661} C_VEL
LIN {X 0,Y 565.025,Z 654.769,A -85,B 0,C 180,E1 26880.764,E2 26880.764} C_VEL
LIN {X 0,Y 565.543,Z 632.214,A -85,B 0,C 180,E1 26880.016,E2 26880.016} C_VEL
LIN {X 0,Y 565.918,Z 610.148,A -85,B 0,C 180,E1 26879.491,E2 26879.491} C_VEL
LIN {X 0,Y 566.232,Z 565.399,A -85,B 0,C 180,E1 26878.821,E2 26878.821} C_VEL
LIN {X 0,Y 567.473,Z 353.357,A -85,B 0,C 180,E1 26875.773,E2 26875.773} C_VEL
LIN {X 0,Y 567.591,Z 311.527,A -85,B 0,C 180,E1 26875.152,E2 26875.152} C_VEL
LIN {X 0,Y 565.81,Z 302.396,A -85,B 0,C 180,E1 26874.861,E2 26874.861} C_VEL
LIN {X 0,Y 566.624,Z 271.734,A -85,B 0,C 180,E1 26872.578,E2 26872.578} C_VEL
LIN {X 0,Y 568.224,Z 271.983,A -85,B 0,C 180,E1 26872.367,E2 26872.367} C_VEL
LIN {X 0,Y 570.828,Z 269.878,A -85,B 0,C 180,E1 26872.03,E2 26872.03} C_VEL
LIN {X 0,Y 574.538,Z 264.171,A -85,B 0,C 180,E1 26871.558,E2 26871.558} C_VEL
LIN {X 0,Y 575.316,Z 262.769,A -85,B 0,C 180,E1 26871.461,E2 26871.461} C_VEL
LIN {X 0,Y 576.409,Z 262.902,A -85,B 0,C 180,E1 26871.325,E2 26871.325} C_VEL
LIN {X 0,Y 576.723,Z 263.291,A -85,B 0,C 180,E1 26871.285,E2 26871.285} C_VEL
LIN {X 0,Y 576.902,Z 337.162,A -85,B 0,C 180,E1 26871.263,E2 26871.263} C_VEL
LIN {X 0,Y 578.072,Z 350.323,A -85,B 0,C 180,E1 26871.119,E2 26871.119} C_VEL
LIN {X 0,Y 580.295,Z 361.726,A -85,B 0,C 180,E1 26870.848,E2 26870.848} C_VEL
LIN {X 0,Y 583.583,Z 371.842,A -85,B 0,C 180,E1 26870.453,E2 26870.453} C_VEL
LIN {X 0,Y 587.818,Z 380.488,A -85,B 0,C 180,E1 26869.954,E2 26869.954} C_VEL
LIN {X 0,Y 590.122,Z 385.1,A -85,B 0,C 180,E1 26869.539,E2 26869.539} C_VEL
LIN {X 0,Y 591.208,Z 388.845,A -85,B 0,C 180,E1 26869.022,E2 26869.022} C_VEL
LIN {X 0,Y 591.027,Z 391.389,A -85,B 0,C 180,E1 26868.458,E2 26868.458} C_VEL
LIN {X 0,Y 589.523,Z 392.788,A -85,B 0,C 180,E1 26867.831,E2 26867.831} C_VEL
LIN {X 0,Y 586.951,Z 392.727,A -85,B 0,C 180,E1 26867.239,E2 26867.239} C_VEL
LIN {X 0,Y 583.725,Z 391.294,A -85,B 0,C 180,E1 26866.717,E2 26866.717} C_VEL
LIN {X 0,Y 578.778,Z 387.349,A -85,B 0,C 180,E1 26866.086,E2 26866.086} C_VEL
LIN {X 0,Y 573.811,Z 381.013,A -85,B 0,C 180,E1 26865.311,E2 26865.311} C_VEL
LIN {X 0,Y 570.298,Z 373.498,A -85,B 0,C 180,E1 26864.53,E2 26864.53} C_VEL
LIN {X 0,Y 567.629,Z 362.414,A -85,B 0,C 180,E1 26863.53,E2 26863.53} C_VEL
LIN {X 0,Y 566.591,Z 349.188,A -85,B 0,C 180,E1 26862.469,E2 26862.469} C_VEL
LIN {X 0,Y 567.766,Z 300.822,A -85,B 0,C 180,E1 26858.824,E2 26858.824} C_VEL
LIN {X 0,Y 568.919,Z 265.353,A -85,B 0,C 180,E1 26856.012,E2 26856.012} C_VEL
LIN {X 0,Y 568.825,Z 261.772,A -85,B 0,C 180,E1 26855.699,E2 26855.699} C_VEL
LIN {X 0,Y 563.692,Z 250.764,A -85,B 0,C 180,E1 26854.214,E2 26854.214} C_VEL
LIN {X 0,Y 561.658,Z 246.542,A -85,B 0,C 180,E1 26853.617,E2 26853.617} C_VEL
LIN {X 0,Y 560.281,Z 242.947,A -85,B 0,C 180,E1 26853.098,E2 26853.098} C_VEL
LIN {X 0,Y 560.258,Z 242.949,A -85,B 0,C 180,E1 26849.744,E2 26849.744} C_VEL
LIN {X 0,Y 560.283,Z 242.97,A -85,B 0,C 180,E1 26846.954,E2 26846.954} C_VEL
LIN {X 0,Y 561.023,Z 247.936,A -85,B 0,C 180,E1 26846.63,E2 26846.63} C_VEL
LIN {X 0,Y 561.599,Z 292.102,A -85,B 0,C 180,E1 26843.837,E2 26843.837} C_VEL
LIN {X 0,Y 561.981,Z 331.355,A -85,B 0,C 180,E1 26841.205,E2 26841.205} C_VEL
LIN {X 0,Y 561.997,Z 366.881,A -85,B 0,C 180,E1 26838.731,E2 26838.731} C_VEL
LIN {X 0,Y 561.712,Z 410.329,A -85,B 0,C 180,E1 26835.635,E2 26835.635} C_VEL
LIN {X 0,Y 561.301,Z 445.479,A -85,B 0,C 180,E1 26833.075,E2 26833.075} C_VEL
LIN {X 0,Y 560.885,Z 485.98,A -85,B 0,C 180,E1 26830.158,E2 26830.158} C_VEL
LIN {X 0,Y 561.219,Z 496.91,A -85,B 0,C 180,E1 26830.008,E2 26830.008} C_VEL
LIN {X 0,Y 560.969,Z 600.131,A -85,B 0,C 180,E1 26828.656,E2 26828.656} C_VEL
LIN {X 0,Y 560.843,Z 614.042,A -85,B 0,C 180,E1 26828.293,E2 26828.293} C_VEL
LIN {X 0,Y 560.7,Z 628.365,A -85,B 0,C 180,E1 26827.737,E2 26827.737} C_VEL
LIN {X 0,Y 560.536,Z 640.694,A -85,B 0,C 180,E1 26827.069,E2 26827.069} C_VEL
LIN {X 0,Y 560.39,Z 652.625,A -85,B 0,C 180,E1 26826.248,E2 26826.248} C_VEL
LIN {X 0,Y 560.235,Z 664.346,A -85,B 0,C 180,E1 26825.203,E2 26825.203} C_VEL
LIN {X 0,Y 560.118,Z 673.368,A -85,B 0,C 180,E1 26824.197,E2 26824.197} C_VEL
LIN {X 0,Y 560.03,Z 682.231,A -85,B 0,C 180,E1 26822.967,E2 26822.967} C_VEL
LIN {X 0,Y 559.966,Z 689.521,A -85,B 0,C 180,E1 26821.637,E2 26821.637} C_VEL
LIN {X 0,Y 559.934,Z 695.072,A -85,B 0,C 180,E1 26820.307,E2 26820.307} C_VEL
LIN {X 0,Y 559.919,Z 699.392,A -85,B 0,C 180,E1 26818.772,E2 26818.772} C_VEL
LIN {X 0,Y 559.918,Z 701.724,A -85,B 0,C 180,E1 26817.338,E2 26817.338} C_VEL
LIN {X 0,Y 559.916,Z 702.444,A -85,B 0,C 180,E1 26815.698,E2 26815.698} C_VEL
LIN {X 0,Y 559.916,Z 701.342,A -85,B 0,C 180,E1 26814.26,E2 26814.26} C_VEL
LIN {X 0,Y 559.923,Z 698.439,A -85,B 0,C 180,E1 26812.716,E2 26812.716} C_VEL
LIN {X 0,Y 559.94,Z 693.798,A -85,B 0,C 180,E1 26811.269,E2 26811.269} C_VEL
LIN {X 0,Y 559.979,Z 687.824,A -85,B 0,C 180,E1 26809.922,E2 26809.922} C_VEL
LIN {X 0,Y 560.05,Z 679.676,A -85,B 0,C 180,E1 26808.562,E2 26808.562} C_VEL
LIN {X 0,Y 560.15,Z 670.96,A -85,B 0,C 180,E1 26807.422,E2 26807.422} C_VEL
LIN {X 0,Y 560.298,Z 659.8,A -85,B 0,C 180,E1 26806.27,E2 26806.27} C_VEL
LIN {X 0,Y 560.424,Z 648.686,A -85,B 0,C 180,E1 26805.372,E2 26805.372} C_VEL
LIN {X 0,Y 560.609,Z 636.504,A -85,B 0,C 180,E1 26804.588,E2 26804.588} C_VEL
LIN {X 0,Y 560.744,Z 622.626,A -85,B 0,C 180,E1 26803.929,E2 26803.929} C_VEL
LIN {X 0,Y 560.883,Z 609.639,A -85,B 0,C 180,E1 26803.484,E2 26803.484} C_VEL
LIN {X 0,Y 560.997,Z 595.166,A -85,B 0,C 180,E1 26803.167,E2 26803.167} C_VEL
LIN {X 0,Y 561.029,Z 577.907,A -85,B 0,C 180,E1 26802.942,E2 26802.942} C_VEL
LIN {X 0,Y 560.072,Z 570.291,A -85,B 0,C 180,E1 26802.821,E2 26802.821} C_VEL
LIN {X 0,Y 554.026,Z 550.306,A -85,B 0,C 180,E1 26802.414,E2 26802.414} C_VEL
LIN {X 0,Y 553.32,Z 543.76,A -85,B 0,C 180,E1 26802.311,E2 26802.311} C_VEL
LIN {X 0,Y 553.229,Z 487.711,A -85,B 0,C 180,E1 26801.576,E2 26801.576} C_VEL
LIN {X 0,Y 553.04,Z 485.536,A -85,B 0,C 180,E1 26801.528,E2 26801.528} C_VEL
LIN {X 0,Y 553.67,Z 440.046,A -85,B 0,C 180,E1 26798.16,E2 26798.16} C_VEL
LIN {X 0,Y 554.061,Z 407.991,A -85,B 0,C 180,E1 26795.817,E2 26795.817} C_VEL
LIN {X 0,Y 554.546,Z 363.444,A -85,B 0,C 180,E1 26792.569,E2 26792.569} C_VEL
LIN {X 0,Y 554.887,Z 321.003,A -85,B 0,C 180,E1 26789.459,E2 26789.459} C_VEL
LIN {X 0,Y 554.954,Z 285.157,A -85,B 0,C 180,E1 26786.851,E2 26786.851} C_VEL
LIN {X 0,Y 555.04,Z 253.148,A -85,B 0,C 180,E1 26784.513,E2 26784.513} C_VEL
LIN {X 0,Y 552.334,Z 243.934,A -85,B 0,C 180,E1 26783.704,E2 26783.704} C_VEL
LIN {X 0,Y 552.311,Z 243.938,A -85,B 0,C 180,E1 26780.414,E2 26780.414} C_VEL
LIN {X 0,Y 552.336,Z 243.937,A -85,B 0,C 180,E1 26777.105,E2 26777.105} C_VEL
LIN {X 0,Y 552.342,Z 243.935,A -85,B 0,C 180,E1 26773.606,E2 26773.606} C_VEL
LIN {X 0,Y 552.332,Z 243.938,A -85,B 0,C 180,E1 26770.188,E2 26770.188} C_VEL
LIN {X 0,Y 552.362,Z 244.081,A -85,B 0,C 180,E1 26769.652,E2 26769.652} C_VEL
LIN {X 0,Y 553.823,Z 247.69,A -85,B 0,C 180,E1 26769.075,E2 26769.075} C_VEL
LIN {X 0,Y 556.818,Z 255.335,A -85,B 0,C 180,E1 26767.888,E2 26767.888} C_VEL
LIN {X 0,Y 558.078,Z 260.276,A -85,B 0,C 180,E1 26767.205,E2 26767.205} C_VEL
LIN {X 0,Y 556.996,Z 278.705,A -85,B 0,C 180,E1 26765.381,E2 26765.381} C_VEL
LIN {X 0,Y 556.505,Z 300.716,A -85,B 0,C 180,E1 26763.426,E2 26763.426} C_VEL
LIN {X 0,Y 558.7,Z 311.638,A -85,B 0,C 180,E1 26763.135,E2 26763.135} C_VEL
LIN {X 0,Y 557.374,Z 544.777,A -85,B 0,C 180,E1 26759.862,E2 26759.862} C_VEL
LIN {X 0,Y 557.113,Z 567.564,A -85,B 0,C 180,E1 26759.474,E2 26759.474} C_VEL
LIN {X 0,Y 556.712,Z 588.336,A -85,B 0,C 180,E1 26758.923,E2 26758.923} C_VEL
LIN {X 0,Y 556.288,Z 607.161,A -85,B 0,C 180,E1 26758.243,E2 26758.243} C_VEL
LIN {X 0,Y 555.727,Z 627.292,A -85,B 0,C 180,E1 26757.31,E2 26757.31} C_VEL
LIN {X 0,Y 555.17,Z 644.832,A -85,B 0,C 180,E1 26756.299,E2 26756.299} C_VEL
LIN {X 0,Y 554.598,Z 662.768,A -85,B 0,C 180,E1 26755.067,E2 26755.067} C_VEL
LIN {X 0,Y 554.003,Z 679.904,A -85,B 0,C 180,E1 26753.651,E2 26753.651} C_VEL
LIN {X 0,Y 553.506,Z 695.164,A -85,B 0,C 180,E1 26752.182,E2 26752.182} C_VEL
LIN {X 0,Y 553.034,Z 709.707,A -85,B 0,C 180,E1 26750.524,E2 26750.524} C_VEL
LIN {X 0,Y 552.678,Z 722.752,A -85,B 0,C 180,E1 26748.786,E2 26748.786} C_VEL
LIN {X 0,Y 552.379,Z 735.077,A -85,B 0,C 180,E1 26746.835,E2 26746.835} C_VEL
LIN {X 0,Y 552.172,Z 744.682,A -85,B 0,C 180,E1 26745.007,E2 26745.007} C_VEL
LIN {X 0,Y 552.035,Z 753.545,A -85,B 0,C 180,E1 26742.979,E2 26742.979} C_VEL
LIN {X 0,Y 551.961,Z 760.573,A -85,B 0,C 180,E1 26740.941,E2 26740.941} C_VEL
LIN {X 0,Y 551.929,Z 766.052,A -85,B 0,C 180,E1 26738.858,E2 26738.858} C_VEL
LIN {X 0,Y 551.916,Z 769.95,A -85,B 0,C 180,E1 26736.658,E2 26736.658} C_VEL
LIN {X 0,Y 551.907,Z 771.973,A -85,B 0,C 180,E1 26734.572,E2 26734.572} C_VEL
LIN {X 0,Y 551.904,Z 772.38,A -85,B 0,C 180,E1 26732.284,E2 26732.284} C_VEL
LIN {X 0,Y 551.918,Z 770.966,A -85,B 0,C 180,E1 26730.104,E2 26730.104} C_VEL
LIN {X 0,Y 551.922,Z 767.591,A -85,B 0,C 180,E1 26727.82,E2 26727.82} C_VEL
LIN {X 0,Y 551.949,Z 763.08,A -85,B 0,C 180,E1 26725.845,E2 26725.845} C_VEL
LIN {X 0,Y 552.011,Z 756.643,A -85,B 0,C 180,E1 26723.761,E2 26723.761} C_VEL
LIN {X 0,Y 552.114,Z 748.73,A -85,B 0,C 180,E1 26721.775,E2 26721.775} C_VEL
LIN {X 0,Y 552.294,Z 739.002,A -85,B 0,C 180,E1 26719.781,E2 26719.781} C_VEL
LIN {X 0,Y 552.542,Z 727.779,A -85,B 0,C 180,E1 26717.883,E2 26717.883} C_VEL
LIN {X 0,Y 552.858,Z 715.988,A -85,B 0,C 180,E1 26716.189,E2 26716.189} C_VEL
LIN {X 0,Y 553.308,Z 701.168,A -85,B 0,C 180,E1 26714.38,E2 26714.38} C_VEL
LIN {X 0,Y 553.789,Z 686.121,A -85,B 0,C 180,E1 26712.831,E2 26712.831} C_VEL
LIN {X 0,Y 554.381,Z 669.047,A -85,B 0,C 180,E1 26711.329,E2 26711.329} C_VEL
LIN {X 0,Y 554.936,Z 652.162,A -85,B 0,C 180,E1 26710.091,E2 26710.091} C_VEL
LIN {X 0,Y 555.528,Z 633.909,A -85,B 0,C 180,E1 26708.957,E2 26708.957} C_VEL
LIN {X 0,Y 556.068,Z 614.451,A -85,B 0,C 180,E1 26707.982,E2 26707.982} C_VEL
LIN {X 0,Y 556.556,Z 596.234,A -85,B 0,C 180,E1 26707.251,E2 26707.251} C_VEL
LIN {X 0,Y 556.993,Z 574.763,A -85,B 0,C 180,E1 26706.602,E2 26706.602} C_VEL
LIN {X 0,Y 557.269,Z 555.368,A -85,B 0,C 180,E1 26706.207,E2 26706.207} C_VEL
LIN {X 0,Y 558.717,Z 314.2,A -85,B 0,C 180,E1 26702.814,E2 26702.814} C_VEL
LIN {X 0,Y 558.5,Z 307.541,A -85,B 0,C 180,E1 26702.704,E2 26702.704} C_VEL
LIN {X 0,Y 556.922,Z 298.815,A -85,B 0,C 180,E1 26702.452,E2 26702.452} C_VEL
LIN {X 0,Y 557.925,Z 262.77,A -85,B 0,C 180,E1 26699.644,E2 26699.644} C_VEL
LIN {X 0,Y 558.025,Z 259.117,A -85,B 0,C 180,E1 26699.324,E2 26699.324} C_VEL
LIN {X 0,Y 555.038,Z 250.586,A -85,B 0,C 180,E1 26698.242,E2 26698.242} C_VEL
LIN {X 0,Y 553.352,Z 246.954,A -85,B 0,C 180,E1 26697.741,E2 26697.741} C_VEL
LIN {X 0,Y 552.322,Z 243.939,A -85,B 0,C 180,E1 26697.33,E2 26697.33} C_VEL
LIN {X 0,Y 552.333,Z 243.941,A -85,B 0,C 180,E1 26693.961,E2 26693.961} C_VEL
LIN {X 0,Y 552.347,Z 243.939,A -85,B 0,C 180,E1 26690.551,E2 26690.551} C_VEL
LIN {X 0,Y 552.334,Z 243.938,A -85,B 0,C 180,E1 26687.105,E2 26687.105} C_VEL
LIN {X 0,Y 552.339,Z 243.936,A -85,B 0,C 180,E1 26683.606,E2 26683.606} C_VEL
LIN {X 0,Y 552.343,Z 243.929,A -85,B 0,C 180,E1 26680.124,E2 26680.124} C_VEL
LIN {X 0,Y 552.318,Z 243.929,A -85,B 0,C 180,E1 26676.814,E2 26676.814} C_VEL
LIN {X 0,Y 552.322,Z 243.937,A -85,B 0,C 180,E1 26673.514,E2 26673.514} C_VEL
LIN {X 0,Y 552.348,Z 243.936,A -85,B 0,C 180,E1 26670.215,E2 26670.215} C_VEL
LIN {X 0,Y 552.342,Z 244.015,A -85,B 0,C 180,E1 26667.768,E2 26667.768} C_VEL
LIN {X 0,Y 555.261,Z 254.313,A -85,B 0,C 180,E1 26666.813,E2 26666.813} C_VEL
LIN {X 0,Y 555.125,Z 299.18,A -85,B 0,C 180,E1 26663.279,E2 26663.279} C_VEL
LIN {X 0,Y 554.846,Z 337.609,A -85,B 0,C 180,E1 26660.243,E2 26660.243} C_VEL
LIN {X 0,Y 554.399,Z 377.948,A -85,B 0,C 180,E1 26657.048,E2 26657.048} C_VEL
LIN {X 0,Y 553.816,Z 416.207,A -85,B 0,C 180,E1 26654.001,E2 26654.001} C_VEL
LIN {X 0,Y 553.556,Z 436.865,A -85,B 0,C 180,E1 26652.372,E2 26652.372} C_VEL
LIN {X 0,Y 554.16,Z 444.751,A -85,B 0,C 180,E1 26652.25,E2 26652.25} C_VEL
LIN {X 0,Y 553.708,Z 577.576,A -85,B 0,C 180,E1 26650.483,E2 26650.483} C_VEL
LIN {X 0,Y 553.56,Z 593.882,A -85,B 0,C 180,E1 26650.091,E2 26650.091} C_VEL
LIN {X 0,Y 553.353,Z 607.963,A -85,B 0,C 180,E1 26649.569,E2 26649.569} C_VEL
LIN {X 0,Y 553.14,Z 620.179,A -85,B 0,C 180,E1 26648.982,E2 26648.982} C_VEL
LIN {X 0,Y 552.912,Z 632.952,A -85,B 0,C 180,E1 26648.214,E2 26648.214} C_VEL
LIN {X 0,Y 552.648,Z 647.24,A -85,B 0,C 180,E1 26647.119,E2 26647.119} C_VEL
LIN {X 0,Y 552.444,Z 657.644,A -85,B 0,C 180,E1 26646.13,E2 26646.13} C_VEL
LIN {X 0,Y 552.267,Z 667.669,A -85,B 0,C 180,E1 26644.986,E2 26644.986} C_VEL
LIN {X 0,Y 552.111,Z 677.945,A -85,B 0,C 180,E1 26643.53,E2 26643.53} C_VEL
LIN {X 0,Y 552.015,Z 685.437,A -85,B 0,C 180,E1 26642.18,E2 26642.18} C_VEL
LIN {X 0,Y 551.957,Z 691.423,A -85,B 0,C 180,E1 26640.831,E2 26640.831} C_VEL
LIN {X 0,Y 551.927,Z 696.917,A -85,B 0,C 180,E1 26639.17,E2 26639.17} C_VEL
LIN {X 0,Y 551.917,Z 700.237,A -85,B 0,C 180,E1 26637.612,E2 26637.612} C_VEL
LIN {X 0,Y 551.915,Z 701.988,A -85,B 0,C 180,E1 26636.157,E2 26636.157} C_VEL
LIN {X 0,Y 551.915,Z 702.426,A -85,B 0,C 180,E1 26634.491,E2 26634.491} C_VEL
LIN {X 0,Y 551.918,Z 701.022,A -85,B 0,C 180,E1 26632.82,E2 26632.82} C_VEL
LIN {X 0,Y 551.92,Z 698.378,A -85,B 0,C 180,E1 26631.352,E2 26631.352} C_VEL
LIN {X 0,Y 551.943,Z 693.998,A -85,B 0,C 180,E1 26629.774,E2 26629.774} C_VEL
LIN {X 0,Y 551.992,Z 687.659,A -85,B 0,C 180,E1 26628.189,E2 26628.189} C_VEL
LIN {X 0,Y 552.064,Z 681.097,A -85,B 0,C 180,E1 26626.916,E2 26626.916} C_VEL
LIN {X 0,Y 552.181,Z 672.994,A -85,B 0,C 180,E1 26625.637,E2 26625.637} C_VEL
LIN {X 0,Y 552.377,Z 661.512,A -85,B 0,C 180,E1 26624.192,E2 26624.192} C_VEL
LIN {X 0,Y 552.571,Z 650.873,A -85,B 0,C 180,E1 26623.117,E2 26623.117} C_VEL
LIN {X 0,Y 552.793,Z 639.275,A -85,B 0,C 180,E1 26622.147,E2 26622.147} C_VEL
LIN {X 0,Y 553.08,Z 624.636,A -85,B 0,C 180,E1 26621.175,E2 26621.175} C_VEL
LIN {X 0,Y 553.286,Z 612.096,A -85,B 0,C 180,E1 26620.524,E2 26620.524} C_VEL
LIN {X 0,Y 553.528,Z 597.517,A -85,B 0,C 180,E1 26619.935,E2 26619.935} C_VEL
LIN {X 0,Y 553.688,Z 581.476,A -85,B 0,C 180,E1 26619.5,E2 26619.5} C_VEL
LIN {X 0,Y 553.816,Z 557.835,A -85,B 0,C 180,E1 26619.142,E2 26619.142} C_VEL
LIN {X 0,Y 553.948,Z 439.983,A -85,B 0,C 180,E1 26617.596,E2 26617.596} C_VEL
LIN {X 0,Y 553.529,Z 436.533,A -85,B 0,C 180,E1 26617.526,E2 26617.526} C_VEL
LIN {X 0,Y 554.144,Z 398.048,A -85,B 0,C 180,E1 26614.445,E2 26614.445} C_VEL
LIN {X 0,Y 554.437,Z 357.553,A -85,B 0,C 180,E1 26611.335,E2 26611.335} C_VEL
LIN {X 0,Y 554.351,Z 325.957,A -85,B 0,C 180,E1 26609.001,E2 26609.001} C_VEL
LIN {X 0,Y 553.917,Z 291.517,A -85,B 0,C 180,E1 26606.553,E2 26606.553} C_VEL
LIN {X 0,Y 552.995,Z 254.358,A -85,B 0,C 180,E1 26604.14,E2 26604.14} C_VEL
LIN {X 0,Y 552.62,Z 245.273,A -85,B 0,C 180,E1 26603.568,E2 26603.568} C_VEL
LIN {X 0,Y 554.841,Z 249.785,A -85,B 0,C 180,E1 26602.995,E2 26602.995} C_VEL
LIN {X 0,Y 562.376,Z 265.162,A -85,B 0,C 180,E1 26601.192,E2 26601.192} C_VEL
LIN {X 0,Y 561.377,Z 317.775,A -85,B 0,C 180,E1 26597.682,E2 26597.682} C_VEL
LIN {X 0,Y 562.947,Z 331.456,A -85,B 0,C 180,E1 26596.649,E2 26596.649} C_VEL
LIN {X 0,Y 565.829,Z 342.083,A -85,B 0,C 180,E1 26595.734,E2 26595.734} C_VEL
LIN {X 0,Y 570.049,Z 350.563,A -85,B 0,C 180,E1 26594.878,E2 26594.878} C_VEL
LIN {X 0,Y 575.17,Z 356.875,A -85,B 0,C 180,E1 26594.115,E2 26594.115} C_VEL
LIN {X 0,Y 581.661,Z 361.902,A -85,B 0,C 180,E1 26593.355,E2 26593.355} C_VEL
LIN {X 0,Y 585.265,Z 363.607,A -85,B 0,C 180,E1 26592.871,E2 26592.871} C_VEL
LIN {X 0,Y 588.189,Z 364.102,A -85,B 0,C 180,E1 26592.312,E2 26592.312} C_VEL
LIN {X 0,Y 589.971,Z 363.419,A -85,B 0,C 180,E1 26591.763,E2 26591.763} C_VEL
LIN {X 0,Y 590.686,Z 361.519,A -85,B 0,C 180,E1 26591.154,E2 26591.154} C_VEL
LIN {X 0,Y 589.971,Z 358.403,A -85,B 0,C 180,E1 26590.569,E2 26590.569} C_VEL
LIN {X 0,Y 587.853,Z 354.363,A -85,B 0,C 180,E1 26590.074,E2 26590.074} C_VEL
LIN {X 0,Y 582.947,Z 346.475,A -85,B 0,C 180,E1 26589.471,E2 26589.471} C_VEL
LIN {X 0,Y 578.719,Z 337.053,A -85,B 0,C 180,E1 26588.96,E2 26588.96} C_VEL
LIN {X 0,Y 575.433,Z 326.167,A -85,B 0,C 180,E1 26588.554,E2 26588.554} C_VEL
LIN {X 0,Y 573.2,Z 314.006,A -85,B 0,C 180,E1 26588.273,E2 26588.273} C_VEL
LIN {X 0,Y 571.978,Z 300.002,A -85,B 0,C 180,E1 26588.118,E2 26588.118} C_VEL
LIN {X 0,Y 571.746,Z 273.257,A -85,B 0,C 180,E1 26588.088,E2 26588.088} C_VEL
LIN {X 0,Y 571.675,Z 270.615,A -85,B 0,C 180,E1 26588.079,E2 26588.079} C_VEL
LIN {X 0,Y 569.944,Z 272.068,A -85,B 0,C 180,E1 26587.856,E2 26587.856} C_VEL
LIN {X 0,Y 565.941,Z 281.279,A -85,B 0,C 180,E1 26587.332,E2 26587.332} C_VEL
LIN {X 0,Y 562.623,Z 286.342,A -85,B 0,C 180,E1 26586.887,E2 26586.887} C_VEL
LIN {X 0,Y 560.978,Z 287.574,A -85,B 0,C 180,E1 26586.662,E2 26586.662} C_VEL
LIN {X 0,Y 559.831,Z 287.531,A -85,B 0,C 180,E1 26586.494,E2 26586.494} C_VEL
LIN {X 0,Y 559.587,Z 302.692,A -85,B 0,C 180,E1 26585.557,E2 26585.557} C_VEL
LIN {X 0,Y 561.195,Z 313.259,A -85,B 0,C 180,E1 26585.277,E2 26585.277} C_VEL
LIN {X 0,Y 559.607,Z 532.832,A -85,B 0,C 180,E1 26582.073,E2 26582.073} C_VEL
LIN {X 0,Y 559.041,Z 609.081,A -85,B 0,C 180,E1 26580.948,E2 26580.948} C_VEL
LIN {X 0,Y 558.587,Z 631.193,A -85,B 0,C 180,E1 26580.426,E2 26580.426} C_VEL
LIN {X 0,Y 558.032,Z 653.462,A -85,B 0,C 180,E1 26579.692,E2 26579.692} C_VEL
LIN {X 0,Y 557.404,Z 674.564,A -85,B 0,C 180,E1 26578.792,E2 26578.792} C_VEL
LIN {X 0,Y 556.675,Z 694.77,A -85,B 0,C 180,E1 26577.723,E2 26577.723} C_VEL
LIN {X 0,Y 555.936,Z 714.646,A -85,B 0,C 180,E1 26576.455,E2 26576.455} C_VEL
LIN {X 0,Y 555.193,Z 733.472,A -85,B 0,C 180,E1 26575.038,E2 26575.038} C_VEL
LIN {X 0,Y 554.459,Z 752.27,A -85,B 0,C 180,E1 26573.374,E2 26573.374} C_VEL
LIN {X 0,Y 553.812,Z 769.341,A -85,B 0,C 180,E1 26571.599,E2 26571.599} C_VEL
LIN {X 0,Y 553.248,Z 785.127,A -85,B 0,C 180,E1 26569.682,E2 26569.682} C_VEL
LIN {X 0,Y 552.812,Z 799.179,A -85,B 0,C 180,E1 26567.69,E2 26567.69} C_VEL
LIN {X 0,Y 552.479,Z 811.526,A -85,B 0,C 180,E1 26565.644,E2 26565.644} C_VEL
LIN {X 0,Y 552.233,Z 822.402,A -85,B 0,C 180,E1 26563.507,E2 26563.507} C_VEL
LIN {X 0,Y 552.076,Z 831.312,A -85,B 0,C 180,E1 26561.386,E2 26561.386} C_VEL
LIN {X 0,Y 551.984,Z 839.175,A -85,B 0,C 180,E1 26559.067,E2 26559.067} C_VEL
LIN {X 0,Y 551.94,Z 844.922,A -85,B 0,C 180,E1 26556.867,E2 26556.867} C_VEL
LIN {X 0,Y 551.918,Z 848.957,A -85,B 0,C 180,E1 26554.676,E2 26554.676} C_VEL
LIN {X 0,Y 551.909,Z 851.561,A -85,B 0,C 180,E1 26552.388,E2 26552.388} C_VEL
LIN {X 0,Y 551.911,Z 852.489,A -85,B 0,C 180,E1 26550.104,E2 26550.104} C_VEL
LIN {X 0,Y 551.912,Z 851.762,A -85,B 0,C 180,E1 26547.924,E2 26547.924} C_VEL
LIN {X 0,Y 551.916,Z 849.431,A -85,B 0,C 180,E1 26545.636,E2 26545.636} C_VEL
LIN {X 0,Y 551.923,Z 845.588,A -85,B 0,C 180,E1 26543.446,E2 26543.446} C_VEL
LIN {X 0,Y 551.958,Z 840.086,A -85,B 0,C 180,E1 26541.248,E2 26541.248} C_VEL
LIN {X 0,Y 552.047,Z 832.821,A -85,B 0,C 180,E1 26539.009,E2 26539.009} C_VEL
LIN {X 0,Y 552.198,Z 823.846,A -85,B 0,C 180,E1 26536.812,E2 26536.812} C_VEL
LIN {X 0,Y 552.429,Z 813.262,A -85,B 0,C 180,E1 26534.677,E2 26534.677} C_VEL
LIN {X 0,Y 552.77,Z 800.593,A -85,B 0,C 180,E1 26532.526,E2 26532.526} C_VEL
LIN {X 0,Y 553.187,Z 787.1,A -85,B 0,C 180,E1 26530.575,E2 26530.575} C_VEL
LIN {X 0,Y 553.707,Z 772.063,A -85,B 0,C 180,E1 26528.712,E2 26528.712} C_VEL
LIN {X 0,Y 554.325,Z 755.613,A -85,B 0,C 180,E1 26526.957,E2 26526.957} C_VEL
LIN {X 0,Y 555.042,Z 737.468,A -85,B 0,C 180,E1 26525.296,E2 26525.296} C_VEL
LIN {X 0,Y 555.757,Z 718.943,A -85,B 0,C 180,E1 26523.846,E2 26523.846} C_VEL
LIN {X 0,Y 556.511,Z 699.63,A -85,B 0,C 180,E1 26522.566,E2 26522.566} C_VEL
LIN {X 0,Y 557.229,Z 679.07,A -85,B 0,C 180,E1 26521.432,E2 26521.432} C_VEL
LIN {X 0,Y 557.885,Z 658.451,A -85,B 0,C 180,E1 26520.5,E2 26520.5} C_VEL
LIN {X 0,Y 558.51,Z 636.237,A -85,B 0,C 180,E1 26519.72,E2 26519.72} C_VEL
LIN {X 0,Y 558.93,Z 613.964,A -85,B 0,C 180,E1 26519.149,E2 26519.149} C_VEL
LIN {X 0,Y 559.276,Z 584.41,A -85,B 0,C 180,E1 26518.669,E2 26518.669} C_VEL
LIN {X 0,Y 560.78,Z 363.98,A -85,B 0,C 180,E1 26515.469,E2 26515.469} C_VEL
LIN {X 0,Y 560.993,Z 312.986,A -85,B 0,C 180,E1 26514.704,E2 26514.704} C_VEL
LIN {X 0,Y 558.916,Z 302.732,A -85,B 0,C 180,E1 26514.387,E2 26514.387} C_VEL
LIN {X 0,Y 559.34,Z 291.95,A -85,B 0,C 180,E1 26513.564,E2 26513.564} C_VEL
LIN {X 0,Y 560.978,Z 292.07,A -85,B 0,C 180,E1 26513.338,E2 26513.338} C_VEL
LIN {X 0,Y 563.676,Z 289.601,A -85,B 0,C 180,E1 26512.971,E2 26512.971} C_VEL
LIN {X 0,Y 567.537,Z 283.237,A -85,B 0,C 180,E1 26512.457,E2 26512.457} C_VEL
LIN {X 0,Y 569.14,Z 279.841,A -85,B 0,C 180,E1 26512.248,E2 26512.248} C_VEL
LIN {X 0,Y 571.755,Z 278.32,A -85,B 0,C 180,E1 26511.911,E2 26511.911} C_VEL
LIN {X 0,Y 571.935,Z 337.57,A -85,B 0,C 180,E1 26511.888,E2 26511.888} C_VEL
LIN {X 0,Y 573.104,Z 351.327,A -85,B 0,C 180,E1 26511.739,E2 26511.739} C_VEL
LIN {X 0,Y 575.316,Z 363.401,A -85,B 0,C 180,E1 26511.461,E2 26511.461} C_VEL
LIN {X 0,Y 578.563,Z 374.198,A -85,B 0,C 180,E1 26511.059,E2 26511.059} C_VEL
LIN {X 0,Y 582.788,Z 383.655,A -85,B 0,C 180,E1 26510.547,E2 26510.547} C_VEL
LIN {X 0,Y 586.451,Z 390.011,A -85,B 0,C 180,E1 26510.065,E2 26510.065} C_VEL
LIN {X 0,Y 588.177,Z 394.191,A -85,B 0,C 180,E1 26509.569,E2 26509.569} C_VEL
LIN {X 0,Y 588.541,Z 397.219,A -85,B 0,C 180,E1 26509.022,E2 26509.022} C_VEL
LIN {X 0,Y 587.615,Z 399.198,A -85,B 0,C 180,E1 26508.424,E2 26508.424} C_VEL
LIN {X 0,Y 585.485,Z 399.936,A -85,B 0,C 180,E1 26507.83,E2 26507.83} C_VEL
LIN {X 0,Y 582.454,Z 399.372,A -85,B 0,C 180,E1 26507.283,E2 26507.283} C_VEL
LIN {X 0,Y 578.804,Z 397.543,A -85,B 0,C 180,E1 26506.801,E2 26506.801} C_VEL
LIN {X 0,Y 572.436,Z 392.302,A -85,B 0,C 180,E1 26506.023,E2 26506.023} C_VEL
LIN {X 0,Y 567.513,Z 385.89,A -85,B 0,C 180,E1 26505.236,E2 26505.236} C_VEL
LIN {X 0,Y 563.577,Z 377.44,A -85,B 0,C 180,E1 26504.347,E2 26504.347} C_VEL
LIN {X 0,Y 560.902,Z 366.446,A -85,B 0,C 180,E1 26503.337,E2 26503.337} C_VEL
LIN {X 0,Y 559.765,Z 353.319,A -85,B 0,C 180,E1 26502.261,E2 26502.261} C_VEL
LIN {X 0,Y 561.22,Z 302.609,A -85,B 0,C 180,E1 26498.381,E2 26498.381} C_VEL
LIN {X 0,Y 562.619,Z 266.434,A -85,B 0,C 180,E1 26495.473,E2 26495.473} C_VEL
LIN {X 0,Y 557.693,Z 255.732,A -85,B 0,C 180,E1 26494.012,E2 26494.012} C_VEL
LIN {X 0,Y 554.059,Z 247.984,A -85,B 0,C 180,E1 26492.9,E2 26492.9} C_VEL
LIN {X 0,Y 552.43,Z 244.562,A -85,B 0,C 180,E1 26492.394,E2 26492.394} C_VEL
LIN {X 0,Y 552.331,Z 243.938,A -85,B 0,C 180,E1 26492.277,E2 26492.277} C_VEL
LIN {X 0,Y 552.342,Z 243.935,A -85,B 0,C 180,E1 26488.903,E2 26488.903} C_VEL
LIN {X 0,Y 552.35,Z 244.098,A -85,B 0,C 180,E1 26487.126,E2 26487.126} C_VEL
LIN {X 0,Y 553.273,Z 249.347,A -85,B 0,C 180,E1 26486.779,E2 26486.779} C_VEL
LIN {X 0,Y 553.852,Z 292.268,A -85,B 0,C 180,E1 26484.078,E2 26484.078} C_VEL
LIN {X 0,Y 554.287,Z 333.664,A -85,B 0,C 180,E1 26481.314,E2 26481.314} C_VEL
LIN {X 0,Y 554.292,Z 373.544,A -85,B 0,C 180,E1 26478.541,E2 26478.541} C_VEL
LIN {X 0,Y 553.923,Z 419.035,A -85,B 0,C 180,E1 26475.28,E2 26475.28} C_VEL
LIN {X 0,Y 553.452,Z 458.306,A -85,B 0,C 180,E1 26472.414,E2 26472.414} C_VEL
LIN {X 0,Y 553.121,Z 486.598,A -85,B 0,C 180,E1 26470.35,E2 26470.35} C_VEL
LIN {X 0,Y 553.453,Z 497.54,A -85,B 0,C 180,E1 26470.199,E2 26470.199} C_VEL
LIN {X 0,Y 553.163,Z 599.95,A -85,B 0,C 180,E1 26468.841,E2 26468.841} C_VEL
LIN {X 0,Y 553.022,Z 613.372,A -85,B 0,C 180,E1 26468.49,E2 26468.49} C_VEL
LIN {X 0,Y 552.865,Z 627.424,A -85,B 0,C 180,E1 26467.952,E2 26467.952} C_VEL
LIN {X 0,Y 552.661,Z 640.539,A -85,B 0,C 180,E1 26467.238,E2 26467.238} C_VEL
LIN {X 0,Y 552.491,Z 651.082,A -85,B 0,C 180,E1 26466.511,E2 26466.511} C_VEL
LIN {X 0,Y 552.317,Z 663.222,A -85,B 0,C 180,E1 26465.453,E2 26465.453} C_VEL
LIN {X 0,Y 552.177,Z 672.15,A -85,B 0,C 180,E1 26464.465,E2 26464.465} C_VEL
LIN {X 0,Y 552.066,Z 680.574,A -85,B 0,C 180,E1 26463.322,E2 26463.322} C_VEL
LIN {X 0,Y 551.984,Z 688.323,A -85,B 0,C 180,E1 26461.972,E2 26461.972} C_VEL
LIN {X 0,Y 551.942,Z 694.113,A -85,B 0,C 180,E1 26460.622,E2 26460.622} C_VEL
LIN {X 0,Y 551.922,Z 698.62,A -85,B 0,C 180,E1 26459.169,E2 26459.169} C_VEL
LIN {X 0,Y 551.917,Z 701.285,A -85,B 0,C 180,E1 26457.715,E2 26457.715} C_VEL
LIN {X 0,Y 551.915,Z 702.375,A -85,B 0,C 180,E1 26456.364,E2 26456.364} C_VEL
LIN {X 0,Y 551.915,Z 702,A -85,B 0,C 180,E1 26454.803,E2 26454.803} C_VEL
LIN {X 0,Y 551.92,Z 699.875,A -85,B 0,C 180,E1 26453.342,E2 26453.342} C_VEL
LIN {X 0,Y 551.928,Z 696.474,A -85,B 0,C 180,E1 26451.981,E2 26451.981} C_VEL
LIN {X 0,Y 551.966,Z 690.526,A -85,B 0,C 180,E1 26450.406,E2 26450.406} C_VEL
LIN {X 0,Y 552.028,Z 683.977,A -85,B 0,C 180,E1 26449.142,E2 26449.142} C_VEL
LIN {X 0,Y 552.137,Z 675.615,A -85,B 0,C 180,E1 26447.874,E2 26447.874} C_VEL
LIN {X 0,Y 552.267,Z 666.127,A -85,B 0,C 180,E1 26446.76,E2 26446.76} C_VEL
LIN {X 0,Y 552.408,Z 656.678,A -85,B 0,C 180,E1 26445.856,E2 26445.856} C_VEL
LIN {X 0,Y 552.593,Z 644.993,A -85,B 0,C 180,E1 26444.95,E2 26444.95} C_VEL
LIN {X 0,Y 552.788,Z 632.414,A -85,B 0,C 180,E1 26444.211,E2 26444.211} C_VEL
LIN {X 0,Y 552.935,Z 620.424,A -85,B 0,C 180,E1 26443.669,E2 26443.669} C_VEL
LIN {X 0,Y 553.114,Z 605.805,A -85,B 0,C 180,E1 26443.198,E2 26443.198} C_VEL
LIN {X 0,Y 553.214,Z 589.579,A -85,B 0,C 180,E1 26442.907,E2 26442.907} C_VEL
LIN {X 0,Y 553.32,Z 543.76,A -85,B 0,C 180,E1 26442.311,E2 26442.311} C_VEL
LIN {X 0,Y 552.377,Z 536.141,A -85,B 0,C 180,E1 26442.189,E2 26442.189} C_VEL
LIN {X 0,Y 546.341,Z 516.148,A -85,B 0,C 180,E1 26441.777,E2 26441.777} C_VEL
LIN {X 0,Y 545.645,Z 509.601,A -85,B 0,C 180,E1 26441.673,E2 26441.673} C_VEL
LIN {X 0,Y 545.451,Z 488.252,A -85,B 0,C 180,E1 26441.381,E2 26441.381} C_VEL
LIN {X 0,Y 545.321,Z 486.615,A -85,B 0,C 180,E1 26441.34,E2 26441.34} C_VEL
LIN {X 0,Y 545.961,Z 443.322,A -85,B 0,C 180,E1 26438.118,E2 26438.118} C_VEL
LIN {X 0,Y 546.542,Z 399.468,A -85,B 0,C 180,E1 26434.901,E2 26434.901} C_VEL
LIN {X 0,Y 547.074,Z 353.413,A -85,B 0,C 180,E1 26431.509,E2 26431.509} C_VEL
LIN {X 0,Y 547.43,Z 311.071,A -85,B 0,C 180,E1 26428.385,E2 26428.385} C_VEL
LIN {X 0,Y 547.63,Z 258.614,A -85,B 0,C 180,E1 26424.564,E2 26424.564} C_VEL
LIN {X 0,Y 547.373,Z 254.967,A -85,B 0,C 180,E1 26424.287,E2 26424.287} C_VEL
LIN {X 0,Y 544.387,Z 244.925,A -85,B 0,C 180,E1 26423.382,E2 26423.382} C_VEL
LIN {X 0,Y 544.392,Z 244.924,A -85,B 0,C 180,E1 26420.134,E2 26420.134} C_VEL
LIN {X 0,Y 544.377,Z 244.928,A -85,B 0,C 180,E1 26416.818,E2 26416.818} C_VEL
LIN {X 0,Y 544.398,Z 244.926,A -85,B 0,C 180,E1 26413.241,E2 26413.241} C_VEL
LIN {X 0,Y 544.373,Z 244.932,A -85,B 0,C 180,E1 26410.5,E2 26410.5} C_VEL
LIN {X 0,Y 545.525,Z 248.118,A -85,B 0,C 180,E1 26409.992,E2 26409.992} C_VEL
LIN {X 0,Y 550.138,Z 258.609,A -85,B 0,C 180,E1 26408.265,E2 26408.265} C_VEL
LIN {X 0,Y 551.568,Z 263.84,A -85,B 0,C 180,E1 26407.524,E2 26407.524} C_VEL
LIN {X 0,Y 549.24,Z 297.158,A -85,B 0,C 180,E1 26404.167,E2 26404.167} C_VEL
LIN {X 0,Y 549.238,Z 300.695,A -85,B 0,C 180,E1 26403.873,E2 26403.873} C_VEL
LIN {X 0,Y 551.775,Z 312.994,A -85,B 0,C 180,E1 26403.533,E2 26403.533} C_VEL
LIN {X 0,Y 550.228,Z 546.808,A -85,B 0,C 180,E1 26400.211,E2 26400.211} C_VEL
LIN {X 0,Y 549.933,Z 568.387,A -85,B 0,C 180,E1 26399.829,E2 26399.829} C_VEL
LIN {X 0,Y 549.47,Z 588.939,A -85,B 0,C 180,E1 26399.27,E2 26399.27} C_VEL
LIN {X 0,Y 548.99,Z 607.371,A -85,B 0,C 180,E1 26398.593,E2 26398.593} C_VEL
LIN {X 0,Y 548.339,Z 627.554,A -85,B 0,C 180,E1 26397.644,E2 26397.644} C_VEL
LIN {X 0,Y 547.743,Z 644.071,A -85,B 0,C 180,E1 26396.683,E2 26396.683} C_VEL
LIN {X 0,Y 547.085,Z 661.774,A -85,B 0,C 180,E1 26395.465,E2 26395.465} C_VEL
LIN {X 0,Y 546.396,Z 678.771,A -85,B 0,C 180,E1 26394.058,E2 26394.058} C_VEL
LIN {X 0,Y 545.823,Z 693.908,A -85,B 0,C 180,E1 26392.593,E2 26392.593} C_VEL
LIN {X 0,Y 545.256,Z 709.261,A -85,B 0,C 180,E1 26390.839,E2 26390.839} C_VEL
LIN {X 0,Y 544.848,Z 721.646,A -85,B 0,C 180,E1 26389.177,E2 26389.177} C_VEL
LIN {X 0,Y 544.486,Z 734.207,A -85,B 0,C 180,E1 26387.197,E2 26387.197} C_VEL
LIN {X 0,Y 544.241,Z 744.089,A -85,B 0,C 180,E1 26385.309,E2 26385.309} C_VEL
LIN {X 0,Y 544.075,Z 752.967,A -85,B 0,C 180,E1 26383.28,E2 26383.28} C_VEL
LIN {X 0,Y 543.979,Z 760.045,A -85,B 0,C 180,E1 26381.235,E2 26381.235} C_VEL
LIN {X 0,Y 543.933,Z 765.179,A -85,B 0,C 180,E1 26379.309,E2 26379.309} C_VEL
LIN {X 0,Y 543.92,Z 769.278,A -85,B 0,C 180,E1 26377.181,E2 26377.181} C_VEL
LIN {X 0,Y 543.912,Z 771.657,A -85,B 0,C 180,E1 26375.062,E2 26375.062} C_VEL
LIN {X 0,Y 543.911,Z 772.479,A -85,B 0,C 180,E1 26372.95,E2 26372.95} C_VEL
LIN {X 0,Y 543.904,Z 771.601,A -85,B 0,C 180,E1 26370.737,E2 26370.737} C_VEL
LIN {X 0,Y 543.909,Z 769.253,A -85,B 0,C 180,E1 26368.736,E2 26368.736} C_VEL
LIN {X 0,Y 543.928,Z 765.286,A -85,B 0,C 180,E1 26366.628,E2 26366.628} C_VEL
LIN {X 0,Y 543.984,Z 759.551,A -85,B 0,C 180,E1 26364.515,E2 26364.515} C_VEL
LIN {X 0,Y 544.08,Z 752.846,A -85,B 0,C 180,E1 26362.609,E2 26362.609} C_VEL
LIN {X 0,Y 544.259,Z 743.567,A -85,B 0,C 180,E1 26360.483,E2 26360.483} C_VEL
LIN {X 0,Y 544.521,Z 732.66,A -85,B 0,C 180,E1 26358.454,E2 26358.454} C_VEL
LIN {X 0,Y 544.918,Z 719.446,A -85,B 0,C 180,E1 26356.416,E2 26356.416} C_VEL
LIN {X 0,Y 545.387,Z 705.82,A -85,B 0,C 180,E1 26354.65,E2 26354.65} C_VEL
LIN {X 0,Y 545.998,Z 689.354,A -85,B 0,C 180,E1 26352.852,E2 26352.852} C_VEL
LIN {X 0,Y 546.642,Z 673.036,A -85,B 0,C 180,E1 26351.348,E2 26351.348} C_VEL
LIN {X 0,Y 547.358,Z 654.414,A -85,B 0,C 180,E1 26349.915,E2 26349.915} C_VEL
LIN {X 0,Y 547.973,Z 637.469,A -85,B 0,C 180,E1 26348.821,E2 26348.821} C_VEL
LIN {X 0,Y 548.667,Z 617.938,A -85,B 0,C 180,E1 26347.783,E2 26347.783} C_VEL
LIN {X 0,Y 549.199,Z 599.634,A -85,B 0,C 180,E1 26347.013,E2 26347.013} C_VEL
LIN {X 0,Y 549.702,Z 579.984,A -85,B 0,C 180,E1 26346.365,E2 26346.365} C_VEL
LIN {X 0,Y 550.085,Z 559.049,A -85,B 0,C 180,E1 26345.895,E2 26345.895} C_VEL
LIN {X 0,Y 551.779,Z 316.662,A -85,B 0,C 180,E1 26342.431,E2 26342.431} C_VEL
LIN {X 0,Y 551.594,Z 308.994,A -85,B 0,C 180,E1 26342.306,E2 26342.306} C_VEL
LIN {X 0,Y 549.742,Z 298.875,A -85,B 0,C 180,E1 26342.015,E2 26342.015} C_VEL
LIN {X 0,Y 550.401,Z 282.478,A -85,B 0,C 180,E1 26340.689,E2 26340.689} C_VEL
LIN {X 0,Y 551.466,Z 262.833,A -85,B 0,C 180,E1 26339.008,E2 26339.008} C_VEL
LIN {X 0,Y 548.545,Z 254.616,A -85,B 0,C 180,E1 26337.95,E2 26337.95} C_VEL
LIN {X 0,Y 545.651,Z 248.361,A -85,B 0,C 180,E1 26337.061,E2 26337.061} C_VEL
LIN {X 0,Y 544.401,Z 244.926,A -85,B 0,C 180,E1 26336.565,E2 26336.565} C_VEL
LIN {X 0,Y 544.393,Z 244.931,A -85,B 0,C 180,E1 26333.088,E2 26333.088} C_VEL
LIN {X 0,Y 544.393,Z 244.928,A -85,B 0,C 180,E1 26329.66,E2 26329.66} C_VEL
LIN {X 0,Y 544.406,Z 244.924,A -85,B 0,C 180,E1 26326.179,E2 26326.179} C_VEL
LIN {X 0,Y 544.379,Z 244.926,A -85,B 0,C 180,E1 26322.811,E2 26322.811} C_VEL
LIN {X 0,Y 544.385,Z 244.926,A -85,B 0,C 180,E1 26319.519,E2 26319.519} C_VEL
LIN {X 0,Y 544.403,Z 244.919,A -85,B 0,C 180,E1 26316.126,E2 26316.126} C_VEL
LIN {X 0,Y 544.403,Z 244.926,A -85,B 0,C 180,E1 26312.682,E2 26312.682} C_VEL
LIN {X 0,Y 544.402,Z 244.925,A -85,B 0,C 180,E1 26309.125,E2 26309.125} C_VEL
LIN {X 0,Y 544.406,Z 245.005,A -85,B 0,C 180,E1 26308.105,E2 26308.105} C_VEL
LIN {X 0,Y 547.78,Z 256.939,A -85,B 0,C 180,E1 26306.98,E2 26306.98} C_VEL
LIN {X 0,Y 547.598,Z 301.426,A -85,B 0,C 180,E1 26303.457,E2 26303.457} C_VEL
LIN {X 0,Y 547.261,Z 341.004,A -85,B 0,C 180,E1 26300.313,E2 26300.313} C_VEL
LIN {X 0,Y 546.738,Z 381.642,A -85,B 0,C 180,E1 26297.069,E2 26297.069} C_VEL
LIN {X 0,Y 546.085,Z 423.618,A -85,B 0,C 180,E1 26293.714,E2 26293.714} C_VEL
LIN {X 0,Y 545.893,Z 437.86,A -85,B 0,C 180,E1 26292.59,E2 26292.59} C_VEL
LIN {X 0,Y 546.463,Z 445.694,A -85,B 0,C 180,E1 26292.467,E2 26292.467} C_VEL
LIN {X 0,Y 545.949,Z 579.205,A -85,B 0,C 180,E1 26290.663,E2 26290.663} C_VEL
LIN {X 0,Y 545.783,Z 595.96,A -85,B 0,C 180,E1 26290.236,E2 26290.236} C_VEL
LIN {X 0,Y 545.567,Z 609.746,A -85,B 0,C 180,E1 26289.707,E2 26289.707} C_VEL
LIN {X 0,Y 545.322,Z 622.41,A -85,B 0,C 180,E1 26289.073,E2 26289.073} C_VEL
LIN {X 0,Y 545.005,Z 637.121,A -85,B 0,C 180,E1 26288.121,E2 26288.121} C_VEL
LIN {X 0,Y 544.737,Z 648.632,A -85,B 0,C 180,E1 26287.17,E2 26287.17} C_VEL
LIN {X 0,Y 544.521,Z 658.339,A -85,B 0,C 180,E1 26286.22,E2 26286.22} C_VEL
LIN {X 0,Y 544.319,Z 668.262,A -85,B 0,C 180,E1 26285.059,E2 26285.059} C_VEL
LIN {X 0,Y 544.137,Z 678.37,A -85,B 0,C 180,E1 26283.582,E2 26283.582} C_VEL
LIN {X 0,Y 544.034,Z 685.28,A -85,B 0,C 180,E1 26282.318,E2 26282.318} C_VEL
LIN {X 0,Y 543.966,Z 691.29,A -85,B 0,C 180,E1 26280.948,E2 26280.948} C_VEL
LIN {X 0,Y 543.93,Z 696.838,A -85,B 0,C 180,E1 26279.263,E2 26279.263} C_VEL
LIN {X 0,Y 543.917,Z 700.179,A -85,B 0,C 180,E1 26277.683,E2 26277.683} C_VEL
LIN {X 0,Y 543.915,Z 701.953,A -85,B 0,C 180,E1 26276.206,E2 26276.206} C_VEL
LIN {X 0,Y 543.914,Z 702.435,A -85,B 0,C 180,E1 26274.515,E2 26274.515} C_VEL
LIN {X 0,Y 543.918,Z 701.059,A -85,B 0,C 180,E1 26272.82,E2 26272.82} C_VEL
LIN {X 0,Y 543.921,Z 698.437,A -85,B 0,C 180,E1 26271.331,E2 26271.331} C_VEL
LIN {X 0,Y 543.948,Z 694.096,A -85,B 0,C 180,E1 26269.73,E2 26269.73} C_VEL
LIN {X 0,Y 544.004,Z 687.796,A -85,B 0,C 180,E1 26268.121,E2 26268.121} C_VEL
LIN {X 0,Y 544.088,Z 681.263,A -85,B 0,C 180,E1 26266.829,E2 26266.829} C_VEL
LIN {X 0,Y 544.224,Z 673.195,A -85,B 0,C 180,E1 26265.531,E2 26265.531} C_VEL
LIN {X 0,Y 544.444,Z 662.286,A -85,B 0,C 180,E1 26264.12,E2 26264.12} C_VEL
LIN {X 0,Y 544.665,Z 651.713,A -85,B 0,C 180,E1 26263.023,E2 26263.023} C_VEL
LIN {X 0,Y 544.927,Z 640.488,A -85,B 0,C 180,E1 26262.046,E2 26262.046} C_VEL
LIN {X 0,Y 545.265,Z 626.34,A -85,B 0,C 180,E1 26261.061,E2 26261.061} C_VEL
LIN {X 0,Y 545.51,Z 612.91,A -85,B 0,C 180,E1 26260.347,E2 26260.347} C_VEL
LIN {X 0,Y 545.762,Z 598.023,A -85,B 0,C 180,E1 26259.742,E2 26259.742} C_VEL
LIN {X 0,Y 545.922,Z 581.641,A -85,B 0,C 180,E1 26259.3,E2 26259.3} C_VEL
LIN {X 0,Y 546.049,Z 552.469,A -85,B 0,C 180,E1 26258.879,E2 26258.879} C_VEL
LIN {X 0,Y 546.205,Z 440.729,A -85,B 0,C 180,E1 26257.392,E2 26257.392} C_VEL
LIN {X 0,Y 545.94,Z 438.274,A -85,B 0,C 180,E1 26257.33,E2 26257.33} C_VEL
LIN {X 0,Y 546.494,Z 399.388,A -85,B 0,C 180,E1 26254.245,E2 26254.245} C_VEL
LIN {X 0,Y 546.788,Z 357.281,A -85,B 0,C 180,E1 26251.015,E2 26251.015} C_VEL
LIN {X 0,Y 546.633,Z 317.175,A -85,B 0,C 180,E1 26248.073,E2 26248.073} C_VEL
LIN {X 0,Y 546.065,Z 287.754,A -85,B 0,C 180,E1 26246.051,E2 26246.051} C_VEL
LIN {X 0,Y 545.236,Z 252.315,A -85,B 0,C 180,E1 26243.762,E2 26243.762} C_VEL
LIN {X 0,Y 546.564,Z 253.75,A -85,B 0,C 180,E1 26243.521,E2 26243.521} C_VEL
LIN {X 0,Y 548.641,Z 254.05,A -85,B 0,C 180,E1 26243.291,E2 26243.291} C_VEL
LIN {X 0,Y 555.899,Z 269.465,A -85,B 0,C 180,E1 26241.482,E2 26241.482} C_VEL
LIN {X 0,Y 554.717,Z 319.638,A -85,B 0,C 180,E1 26238.11,E2 26238.11} C_VEL
LIN {X 0,Y 556.156,Z 333.871,A -85,B 0,C 180,E1 26237.03,E2 26237.03} C_VEL
LIN {X 0,Y 559,Z 345.225,A -85,B 0,C 180,E1 26236.053,E2 26236.053} C_VEL
LIN {X 0,Y 563.04,Z 354.075,A -85,B 0,C 180,E1 26235.171,E2 26235.171} C_VEL
LIN {X 0,Y 568.545,Z 361.507,A -85,B 0,C 180,E1 26234.295,E2 26234.295} C_VEL
LIN {X 0,Y 574.88,Z 366.987,A -85,B 0,C 180,E1 26233.509,E2 26233.509} C_VEL
LIN {X 0,Y 580.293,Z 370.1,A -85,B 0,C 180,E1 26232.922,E2 26232.922} C_VEL
LIN {X 0,Y 583.771,Z 371.206,A -85,B 0,C 180,E1 26232.422,E2 26232.422} C_VEL
LIN {X 0,Y 586.491,Z 371.147,A -85,B 0,C 180,E1 26231.841,E2 26231.841} C_VEL
LIN {X 0,Y 587.965,Z 369.97,A -85,B 0,C 180,E1 26231.268,E2 26231.268} C_VEL
LIN {X 0,Y 588.197,Z 367.624,A -85,B 0,C 180,E1 26230.663,E2 26230.663} C_VEL
LIN {X 0,Y 586.99,Z 364.289,A -85,B 0,C 180,E1 26230.11,E2 26230.11} C_VEL
LIN {X 0,Y 584.374,Z 360.075,A -85,B 0,C 180,E1 26229.642,E2 26229.642} C_VEL
LIN {X 0,Y 578.994,Z 351.476,A -85,B 0,C 180,E1 26228.994,E2 26228.994} C_VEL
LIN {X 0,Y 574.577,Z 341.573,A -85,B 0,C 180,E1 26228.447,E2 26228.447} C_VEL
LIN {X 0,Y 571.097,Z 330.221,A -85,B 0,C 180,E1 26228.005,E2 26228.005} C_VEL
LIN {X 0,Y 568.643,Z 317.542,A -85,B 0,C 180,E1 26227.687,E2 26227.687} C_VEL
LIN {X 0,Y 567.232,Z 303.363,A -85,B 0,C 180,E1 26227.503,E2 26227.503} C_VEL
LIN {X 0,Y 566.776,Z 291.172,A -85,B 0,C 180,E1 26227.442,E2 26227.442} C_VEL
LIN {X 0,Y 563.525,Z 294.586,A -85,B 0,C 180,E1 26227.009,E2 26227.009} C_VEL
LIN {X 0,Y 562.623,Z 295.469,A -85,B 0,C 180,E1 26226.887,E2 26226.887} C_VEL
LIN {X 0,Y 558.228,Z 306.503,A -85,B 0,C 180,E1 26226.281,E2 26226.281} C_VEL
LIN {X 0,Y 556.385,Z 311.535,A -85,B 0,C 180,E1 26226.022,E2 26226.022} C_VEL
LIN {X 0,Y 555.065,Z 313.002,A -85,B 0,C 180,E1 26225.834,E2 26225.834} C_VEL
LIN {X 0,Y 554.618,Z 313.232,A -85,B 0,C 180,E1 26225.76,E2 26225.76} C_VEL
LIN {X 0,Y 552.912,Z 523.162,A -85,B 0,C 180,E1 26222.654,E2 26222.654} C_VEL
LIN {X 0,Y 552.179,Z 608.892,A -85,B 0,C 180,E1 26221.38,E2 26221.38} C_VEL
LIN {X 0,Y 551.654,Z 631.012,A -85,B 0,C 180,E1 26220.856,E2 26220.856} C_VEL
LIN {X 0,Y 551.035,Z 653.323,A -85,B 0,C 180,E1 26220.114,E2 26220.114} C_VEL
LIN {X 0,Y 550.289,Z 674.56,A -85,B 0,C 180,E1 26219.2,E2 26219.2} C_VEL
LIN {X 0,Y 549.466,Z 694.778,A -85,B 0,C 180,E1 26218.119,E2 26218.119} C_VEL
LIN {X 0,Y 548.592,Z 714.975,A -85,B 0,C 180,E1 26216.814,E2 26216.814} C_VEL
LIN {X 0,Y 547.722,Z 733.942,A -85,B 0,C 180,E1 26215.363,E2 26215.363} C_VEL
LIN {X 0,Y 546.9,Z 752.27,A -85,B 0,C 180,E1 26213.717,E2 26213.717} C_VEL
LIN {X 0,Y 546.12,Z 770.043,A -85,B 0,C 180,E1 26211.839,E2 26211.839} C_VEL
LIN {X 0,Y 545.447,Z 786.284,A -85,B 0,C 180,E1 26209.824,E2 26209.824} C_VEL
LIN {X 0,Y 544.929,Z 800.597,A -85,B 0,C 180,E1 26207.733,E2 26207.733} C_VEL
LIN {X 0,Y 544.529,Z 813.266,A -85,B 0,C 180,E1 26205.55,E2 26205.55} C_VEL
LIN {X 0,Y 544.243,Z 824.312,A -85,B 0,C 180,E1 26203.276,E2 26203.276} C_VEL
LIN {X 0,Y 544.065,Z 833.314,A -85,B 0,C 180,E1 26201.019,E2 26201.019} C_VEL
LIN {X 0,Y 543.966,Z 840.393,A -85,B 0,C 180,E1 26198.775,E2 26198.775} C_VEL
LIN {X 0,Y 543.922,Z 846.007,A -85,B 0,C 180,E1 26196.438,E2 26196.438} C_VEL
LIN {X 0,Y 543.915,Z 849.737,A -85,B 0,C 180,E1 26194.217,E2 26194.217} C_VEL
LIN {X 0,Y 543.907,Z 851.898,A -85,B 0,C 180,E1 26191.896,E2 26191.896} C_VEL
LIN {X 0,Y 543.897,Z 852.439,A -85,B 0,C 180,E1 26189.579,E2 26189.579} C_VEL
LIN {X 0,Y 543.908,Z 851.332,A -85,B 0,C 180,E1 26187.26,E2 26187.26} C_VEL
LIN {X 0,Y 543.921,Z 848.483,A -85,B 0,C 180,E1 26184.938,E2 26184.938} C_VEL
LIN {X 0,Y 543.941,Z 843.932,A -85,B 0,C 180,E1 26182.607,E2 26182.607} C_VEL
LIN {X 0,Y 544.002,Z 837.925,A -85,B 0,C 180,E1 26180.372,E2 26180.372} C_VEL
LIN {X 0,Y 544.12,Z 830.092,A -85,B 0,C 180,E1 26178.123,E2 26178.123} C_VEL
LIN {X 0,Y 544.328,Z 820.35,A -85,B 0,C 180,E1 26175.859,E2 26175.859} C_VEL
LIN {X 0,Y 544.647,Z 809.119,A -85,B 0,C 180,E1 26173.687,E2 26173.687} C_VEL
LIN {X 0,Y 545.07,Z 796.341,A -85,B 0,C 180,E1 26171.608,E2 26171.608} C_VEL
LIN {X 0,Y 545.606,Z 782.039,A -85,B 0,C 180,E1 26169.623,E2 26169.623} C_VEL
LIN {X 0,Y 546.283,Z 765.96,A -85,B 0,C 180,E1 26167.707,E2 26167.707} C_VEL
LIN {X 0,Y 547.06,Z 748.73,A -85,B 0,C 180,E1 26165.947,E2 26165.947} C_VEL
LIN {X 0,Y 547.918,Z 730.04,A -85,B 0,C 180,E1 26164.316,E2 26164.316} C_VEL
LIN {X 0,Y 548.769,Z 710.945,A -85,B 0,C 180,E1 26162.903,E2 26162.903} C_VEL
LIN {X 0,Y 549.627,Z 690.798,A -85,B 0,C 180,E1 26161.653,E2 26161.653} C_VEL
LIN {X 0,Y 550.452,Z 669.656,A -85,B 0,C 180,E1 26160.571,E2 26160.571} C_VEL
LIN {X 0,Y 551.203,Z 648.458,A -85,B 0,C 180,E1 26159.705,E2 26159.705} C_VEL
LIN {X 0,Y 551.789,Z 626.471,A -85,B 0,C 180,E1 26159.02,E2 26159.02} C_VEL
LIN {X 0,Y 552.242,Z 604.503,A -85,B 0,C 180,E1 26158.542,E2 26158.542} C_VEL
LIN {X 0,Y 554.068,Z 379.057,A -85,B 0,C 180,E1 26155.223,E2 26155.223} C_VEL
LIN {X 0,Y 554.481,Z 314.71,A -85,B 0,C 180,E1 26154.25,E2 26154.25} C_VEL
LIN {X 0,Y 555.798,Z 314.03,A -85,B 0,C 180,E1 26154.061,E2 26154.061} C_VEL
LIN {X 0,Y 557.564,Z 310.464,A -85,B 0,C 180,E1 26153.812,E2 26153.812} C_VEL
LIN {X 0,Y 559.191,Z 305.54,A -85,B 0,C 180,E1 26153.585,E2 26153.585} C_VEL
LIN {X 0,Y 561.874,Z 299.928,A -85,B 0,C 180,E1 26153.215,E2 26153.215} C_VEL
LIN {X 0,Y 565.033,Z 297.745,A -85,B 0,C 180,E1 26152.789,E2 26152.789} C_VEL
LIN {X 0,Y 566.858,Z 295.645,A -85,B 0,C 180,E1 26152.547,E2 26152.547} C_VEL
LIN {X 0,Y 567.047,Z 338.198,A -85,B 0,C 180,E1 26152.522,E2 26152.522} C_VEL
LIN {X 0,Y 568.224,Z 352.453,A -85,B 0,C 180,E1 26152.367,E2 26152.367} C_VEL
LIN {X 0,Y 570.444,Z 365.199,A -85,B 0,C 180,E1 26152.079,E2 26152.079} C_VEL
LIN {X 0,Y 573.724,Z 376.772,A -85,B 0,C 180,E1 26151.661,E2 26151.661} C_VEL
LIN {X 0,Y 577.973,Z 386.964,A -85,B 0,C 180,E1 26151.131,E2 26151.131} C_VEL
LIN {X 0,Y 583.042,Z 395.719,A -85,B 0,C 180,E1 26150.503,E2 26150.503} C_VEL
LIN {X 0,Y 585.16,Z 400.052,A -85,B 0,C 180,E1 26150.023,E2 26150.023} C_VEL
LIN {X 0,Y 585.872,Z 403.218,A -85,B 0,C 180,E1 26149.506,E2 26149.506} C_VEL
LIN {X 0,Y 585.479,Z 405.288,A -85,B 0,C 180,E1 26149.01,E2 26149.01} C_VEL
LIN {X 0,Y 583.942,Z 406.635,A -85,B 0,C 180,E1 26148.439,E2 26148.439} C_VEL
LIN {X 0,Y 581.194,Z 406.848,A -85,B 0,C 180,E1 26147.857,E2 26147.857} C_VEL
LIN {X 0,Y 577.74,Z 405.832,A -85,B 0,C 180,E1 26147.351,E2 26147.351} C_VEL
LIN {X 0,Y 571.715,Z 402.245,A -85,B 0,C 180,E1 26146.679,E2 26146.679} C_VEL
LIN {X 0,Y 565.523,Z 396.597,A -85,B 0,C 180,E1 26145.874,E2 26145.874} C_VEL
LIN {X 0,Y 560.245,Z 389.078,A -85,B 0,C 180,E1 26144.969,E2 26144.969} C_VEL
LIN {X 0,Y 556.503,Z 380.29,A -85,B 0,C 180,E1 26144.052,E2 26144.052} C_VEL
LIN {X 0,Y 553.869,Z 368.392,A -85,B 0,C 180,E1 26142.958,E2 26142.958} C_VEL
LIN {X 0,Y 552.912,Z 354.152,A -85,B 0,C 180,E1 26141.788,E2 26141.788} C_VEL
LIN {X 0,Y 554.66,Z 305.618,A -85,B 0,C 180,E1 26138.023,E2 26138.023} C_VEL
LIN {X 0,Y 556.208,Z 270.632,A -85,B 0,C 180,E1 26135.179,E2 26135.179} C_VEL
LIN {X 0,Y 551.707,Z 260.686,A -85,B 0,C 180,E1 26133.805,E2 26133.805} C_VEL
LIN {X 0,Y 547.69,Z 252.447,A -85,B 0,C 180,E1 26132.585,E2 26132.585} C_VEL
LIN {X 0,Y 546.12,Z 248.967,A -85,B 0,C 180,E1 26132.069,E2 26132.069} C_VEL
LIN {X 0,Y 544.514,Z 245.646,A -85,B 0,C 180,E1 26131.555,E2 26131.555} C_VEL
LIN {X 0,Y 544.392,Z 244.926,A -85,B 0,C 180,E1 26131.44,E2 26131.44} C_VEL
LIN {X 0,Y 544.378,Z 244.923,A -85,B 0,C 180,E1 26128.047,E2 26128.047} C_VEL
LIN {X 0,Y 544.383,Z 244.987,A -85,B 0,C 180,E1 26127.333,E2 26127.333} C_VEL
LIN {X 0,Y 545.553,Z 250.303,A -85,B 0,C 180,E1 26126.975,E2 26126.975} C_VEL
LIN {X 0,Y 546.117,Z 292.464,A -85,B 0,C 180,E1 26124.326,E2 26124.326} C_VEL
LIN {X 0,Y 546.569,Z 332.373,A -85,B 0,C 180,E1 26121.672,E2 26121.672} C_VEL
LIN {X 0,Y 546.622,Z 372.583,A -85,B 0,C 180,E1 26118.89,E2 26118.89} C_VEL
LIN {X 0,Y 546.27,Z 420.062,A -85,B 0,C 180,E1 26115.499,E2 26115.499} C_VEL
LIN {X 0,Y 545.735,Z 464.183,A -85,B 0,C 180,E1 26112.27,E2 26112.27} C_VEL
LIN {X 0,Y 545.436,Z 488.21,A -85,B 0,C 180,E1 26110.522,E2 26110.522} C_VEL
LIN {X 0,Y 545.58,Z 524.644,A -85,B 0,C 180,E1 26110.033,E2 26110.033} C_VEL
LIN {X 0,Y 545.337,Z 601.547,A -85,B 0,C 180,E1 26108.989,E2 26108.989} C_VEL
LIN {X 0,Y 545.196,Z 616.075,A -85,B 0,C 180,E1 26108.596,E2 26108.596} C_VEL
LIN {X 0,Y 545.016,Z 630.165,A -85,B 0,C 180,E1 26108.014,E2 26108.014} C_VEL
LIN {X 0,Y 544.809,Z 642.257,A -85,B 0,C 180,E1 26107.328,E2 26107.328} C_VEL
LIN {X 0,Y 544.603,Z 653.899,A -85,B 0,C 180,E1 26106.483,E2 26106.483} C_VEL
LIN {X 0,Y 544.382,Z 664.957,A -85,B 0,C 180,E1 26105.442,E2 26105.442} C_VEL
LIN {X 0,Y 544.214,Z 673.615,A -85,B 0,C 180,E1 26104.425,E2 26104.425} C_VEL
LIN {X 0,Y 544.075,Z 682.32,A -85,B 0,C 180,E1 26103.16,E2 26103.16} C_VEL
LIN {X 0,Y 543.987,Z 689.076,A -85,B 0,C 180,E1 26101.896,E2 26101.896} C_VEL
LIN {X 0,Y 543.945,Z 694.324,A -85,B 0,C 180,E1 26100.632,E2 26100.632} C_VEL
LIN {X 0,Y 543.923,Z 698.763,A -85,B 0,C 180,E1 26099.157,E2 26099.157} C_VEL
LIN {X 0,Y 543.917,Z 701.346,A -85,B 0,C 180,E1 26097.682,E2 26097.682} C_VEL
LIN {X 0,Y 543.915,Z 702.389,A -85,B 0,C 180,E1 26096.311,E2 26096.311} C_VEL
LIN {X 0,Y 543.916,Z 701.936,A -85,B 0,C 180,E1 26094.726,E2 26094.726} C_VEL
LIN {X 0,Y 543.92,Z 699.747,A -85,B 0,C 180,E1 26093.243,E2 26093.243} C_VEL
LIN {X 0,Y 543.933,Z 696.296,A -85,B 0,C 180,E1 26091.863,E2 26091.863} C_VEL
LIN {X 0,Y 543.974,Z 690.731,A -85,B 0,C 180,E1 26090.371,E2 26090.371} C_VEL
LIN {X 0,Y 544.036,Z 684.834,A -85,B 0,C 180,E1 26089.195,E2 26089.195} C_VEL
LIN {X 0,Y 544.143,Z 677.461,A -85,B 0,C 180,E1 26088.016,E2 26088.016} C_VEL
LIN {X 0,Y 544.329,Z 667.276,A -85,B 0,C 180,E1 26086.726,E2 26086.726} C_VEL
LIN {X 0,Y 544.511,Z 657.53,A -85,B 0,C 180,E1 26085.755,E2 26085.755} C_VEL
LIN {X 0,Y 544.728,Z 646.051,A -85,B 0,C 180,E1 26084.837,E2 26084.837} C_VEL
LIN {X 0,Y 544.956,Z 633.5,A -85,B 0,C 180,E1 26084.074,E2 26084.074} C_VEL
LIN {X 0,Y 545.13,Z 620.633,A -85,B 0,C 180,E1 26083.483,E2 26083.483} C_VEL
LIN {X 0,Y 545.309,Z 605.1,A -85,B 0,C 180,E1 26082.998,E2 26082.998} C_VEL
LIN {X 0,Y 545.398,Z 588.568,A -85,B 0,C 180,E1 26082.716,E2 26082.716} C_VEL
LIN {X 0,Y 545.645,Z 509.601,A -85,B 0,C 180,E1 26081.673,E2 26081.673} C_VEL
LIN {X 0,Y 544.708,Z 503.65,A -85,B 0,C 180,E1 26081.554,E2 26081.554} C_VEL
LIN {X 0,Y 539.945,Z 493.422,A -85,B 0,C 180,E1 26081.301,E2 26081.301} C_VEL
LIN {X 0,Y 537.614,Z 487.564,A -85,B 0,C 180,E1 26081.135,E2 26081.135} C_VEL
LIN {X 0,Y 538.265,Z 445.858,A -85,B 0,C 180,E1 26078.019,E2 26078.019} C_VEL
LIN {X 0,Y 538.932,Z 399.31,A -85,B 0,C 180,E1 26074.579,E2 26074.579} C_VEL
LIN {X 0,Y 539.495,Z 353.553,A -85,B 0,C 180,E1 26071.192,E2 26071.192} C_VEL
LIN {X 0,Y 539.872,Z 309.706,A -85,B 0,C 180,E1 26067.953,E2 26067.953} C_VEL
LIN {X 0,Y 540.158,Z 258.343,A -85,B 0,C 180,E1 26064.191,E2 26064.191} C_VEL
LIN {X 0,Y 536.455,Z 245.916,A -85,B 0,C 180,E1 26063.059,E2 26063.059} C_VEL
LIN {X 0,Y 536.455,Z 245.914,A -85,B 0,C 180,E1 26059.668,E2 26059.668} C_VEL
LIN {X 0,Y 536.428,Z 245.917,A -85,B 0,C 180,E1 26056.397,E2 26056.397} C_VEL
LIN {X 0,Y 536.462,Z 245.915,A -85,B 0,C 180,E1 26053.012,E2 26053.012} C_VEL
LIN {X 0,Y 536.47,Z 246.06,A -85,B 0,C 180,E1 26051.346,E2 26051.346} C_VEL
LIN {X 0,Y 537.664,Z 249.297,A -85,B 0,C 180,E1 26050.81,E2 26050.81} C_VEL
LIN {X 0,Y 541.934,Z 258.652,A -85,B 0,C 180,E1 26049.204,E2 26049.204} C_VEL
LIN {X 0,Y 544.403,Z 265.099,A -85,B 0,C 180,E1 26048.179,E2 26048.179} C_VEL
LIN {X 0,Y 545.008,Z 267.958,A -85,B 0,C 180,E1 26047.789,E2 26047.789} C_VEL
LIN {X 0,Y 542.509,Z 299.775,A -85,B 0,C 180,E1 26044.529,E2 26044.529} C_VEL
LIN {X 0,Y 542.455,Z 302.354,A -85,B 0,C 180,E1 26044.299,E2 26044.299} C_VEL
LIN {X 0,Y 544.876,Z 314.529,A -85,B 0,C 180,E1 26043.94,E2 26043.94} C_VEL
LIN {X 0,Y 543.099,Z 549.622,A -85,B 0,C 180,E1 26040.558,E2 26040.558} C_VEL
LIN {X 0,Y 542.755,Z 570.771,A -85,B 0,C 180,E1 26040.159,E2 26040.159} C_VEL
LIN {X 0,Y 542.226,Z 590.19,A -85,B 0,C 180,E1 26039.605,E2 26039.605} C_VEL
LIN {X 0,Y 541.674,Z 609.086,A -85,B 0,C 180,E1 26038.892,E2 26038.892} C_VEL
LIN {X 0,Y 540.923,Z 628.935,A -85,B 0,C 180,E1 26037.925,E2 26037.925} C_VEL
LIN {X 0,Y 540.266,Z 645.105,A -85,B 0,C 180,E1 26036.963,E2 26036.963} C_VEL
LIN {X 0,Y 539.506,Z 663.018,A -85,B 0,C 180,E1 26035.701,E2 26035.701} C_VEL
LIN {X 0,Y 538.729,Z 679.751,A -85,B 0,C 180,E1 26034.28,E2 26034.28} C_VEL
LIN {X 0,Y 538.103,Z 694.408,A -85,B 0,C 180,E1 26032.834,E2 26032.834} C_VEL
LIN {X 0,Y 537.45,Z 709.759,A -85,B 0,C 180,E1 26031.042,E2 26031.042} C_VEL
LIN {X 0,Y 536.984,Z 722.088,A -85,B 0,C 180,E1 26029.356,E2 26029.356} C_VEL
LIN {X 0,Y 536.567,Z 734.559,A -85,B 0,C 180,E1 26027.347,E2 26027.347} C_VEL
LIN {X 0,Y 536.292,Z 744.335,A -85,B 0,C 180,E1 26025.442,E2 26025.442} C_VEL
LIN {X 0,Y 536.1,Z 753.21,A -85,B 0,C 180,E1 26023.372,E2 26023.372} C_VEL
LIN {X 0,Y 535.988,Z 760.226,A -85,B 0,C 180,E1 26021.296,E2 26021.296} C_VEL
LIN {X 0,Y 535.937,Z 765.327,A -85,B 0,C 180,E1 26019.341,E2 26019.341} C_VEL
LIN {X 0,Y 535.922,Z 769.533,A -85,B 0,C 180,E1 26017.073,E2 26017.073} C_VEL
LIN {X 0,Y 535.915,Z 771.774,A -85,B 0,C 180,E1 26014.923,E2 26014.923} C_VEL
LIN {X 0,Y 535.907,Z 772.49,A -85,B 0,C 180,E1 26012.781,E2 26012.781} C_VEL
LIN {X 0,Y 535.901,Z 771.442,A -85,B 0,C 180,E1 26010.535,E2 26010.535} C_VEL
LIN {X 0,Y 535.908,Z 769.002,A -85,B 0,C 180,E1 26008.503,E2 26008.503} C_VEL
LIN {X 0,Y 535.944,Z 764.637,A -85,B 0,C 180,E1 26006.256,E2 26006.256} C_VEL
LIN {X 0,Y 536.013,Z 758.675,A -85,B 0,C 180,E1 26004.111,E2 26004.111} C_VEL
LIN {X 0,Y 536.142,Z 750.946,A -85,B 0,C 180,E1 26001.96,E2 26001.96} C_VEL
LIN {X 0,Y 536.353,Z 741.649,A -85,B 0,C 180,E1 25999.908,E2 25999.908} C_VEL
LIN {X 0,Y 536.676,Z 731.03,A -85,B 0,C 180,E1 25997.956,E2 25997.956} C_VEL
LIN {X 0,Y 537.118,Z 718.209,A -85,B 0,C 180,E1 25995.995,E2 25995.995} C_VEL
LIN {X 0,Y 537.66,Z 704.755,A -85,B 0,C 180,E1 25994.246,E2 25994.246} C_VEL
LIN {X 0,Y 538.337,Z 688.706,A -85,B 0,C 180,E1 25992.489,E2 25992.489} C_VEL
LIN {X 0,Y 539.066,Z 672.741,A -85,B 0,C 180,E1 25991.003,E2 25991.003} C_VEL
LIN {X 0,Y 539.873,Z 654.4,A -85,B 0,C 180,E1 25989.576,E2 25989.576} C_VEL
LIN {X 0,Y 540.551,Z 637.945,A -85,B 0,C 180,E1 25988.499,E2 25988.499} C_VEL
LIN {X 0,Y 541.338,Z 618.515,A -85,B 0,C 180,E1 25987.446,E2 25987.446} C_VEL
LIN {X 0,Y 541.939,Z 600.312,A -85,B 0,C 180,E1 25986.667,E2 25986.667} C_VEL
LIN {X 0,Y 542.458,Z 582.195,A -85,B 0,C 180,E1 25986.053,E2 25986.053} C_VEL
LIN {X 0,Y 542.941,Z 560.37,A -85,B 0,C 180,E1 25985.534,E2 25985.534} C_VEL
LIN {X 0,Y 543.565,Z 483.05,A -85,B 0,C 180,E1 25984.401,E2 25984.401} C_VEL
LIN {X 0,Y 544.777,Z 310.759,A -85,B 0,C 180,E1 25981.907,E2 25981.907} C_VEL
LIN {X 0,Y 542.906,Z 300.459,A -85,B 0,C 180,E1 25981.6,E2 25981.6} C_VEL
LIN {X 0,Y 545.044,Z 266.838,A -85,B 0,C 180,E1 25978.724,E2 25978.724} C_VEL
LIN {X 0,Y 541.922,Z 258.073,A -85,B 0,C 180,E1 25977.576,E2 25977.576} C_VEL
LIN {X 0,Y 537.557,Z 249.084,A -85,B 0,C 180,E1 25976.246,E2 25976.246} C_VEL
LIN {X 0,Y 536.445,Z 245.917,A -85,B 0,C 180,E1 25975.809,E2 25975.809} C_VEL
LIN {X 0,Y 536.468,Z 245.917,A -85,B 0,C 180,E1 25972.449,E2 25972.449} C_VEL
LIN {X 0,Y 536.451,Z 245.917,A -85,B 0,C 180,E1 25969.013,E2 25969.013} C_VEL
LIN {X 0,Y 536.451,Z 245.914,A -85,B 0,C 180,E1 25965.55,E2 25965.55} C_VEL
LIN {X 0,Y 536.459,Z 245.913,A -85,B 0,C 180,E1 25962.115,E2 25962.115} C_VEL
LIN {X 0,Y 536.465,Z 245.914,A -85,B 0,C 180,E1 25958.637,E2 25958.637} C_VEL
LIN {X 0,Y 536.463,Z 245.914,A -85,B 0,C 180,E1 25955.034,E2 25955.034} C_VEL
LIN {X 0,Y 536.461,Z 245.915,A -85,B 0,C 180,E1 25951.458,E2 25951.458} C_VEL
LIN {X 0,Y 536.466,Z 246.081,A -85,B 0,C 180,E1 25948.438,E2 25948.438} C_VEL
LIN {X 0,Y 540.335,Z 259.081,A -85,B 0,C 180,E1 25947.198,E2 25947.198} C_VEL
LIN {X 0,Y 540.073,Z 304.266,A -85,B 0,C 180,E1 25943.592,E2 25943.592} C_VEL
LIN {X 0,Y 539.674,Z 344.607,A -85,B 0,C 180,E1 25940.368,E2 25940.368} C_VEL
LIN {X 0,Y 539.077,Z 386.822,A -85,B 0,C 180,E1 25936.986,E2 25936.986} C_VEL
LIN {X 0,Y 538.367,Z 429.073,A -85,B 0,C 180,E1 25933.588,E2 25933.588} C_VEL
LIN {X 0,Y 538.266,Z 439.033,A -85,B 0,C 180,E1 25932.813,E2 25932.813} C_VEL
LIN {X 0,Y 538.774,Z 446.515,A -85,B 0,C 180,E1 25932.692,E2 25932.692} C_VEL
LIN {X 0,Y 538.179,Z 580.948,A -85,B 0,C 180,E1 25930.839,E2 25930.839} C_VEL
LIN {X 0,Y 538.01,Z 598.017,A -85,B 0,C 180,E1 25930.386,E2 25930.386} C_VEL
LIN {X 0,Y 537.775,Z 612.757,A -85,B 0,C 180,E1 25929.799,E2 25929.799} C_VEL
LIN {X 0,Y 537.48,Z 627.811,A -85,B 0,C 180,E1 25928.99,E2 25928.99} C_VEL
LIN {X 0,Y 537.151,Z 640.781,A -85,B 0,C 180,E1 25928.079,E2 25928.079} C_VEL
LIN {X 0,Y 536.854,Z 653.082,A -85,B 0,C 180,E1 25927.007,E2 25927.007} C_VEL
LIN {X 0,Y 536.536,Z 665.269,A -85,B 0,C 180,E1 25925.669,E2 25925.669} C_VEL
LIN {X 0,Y 536.297,Z 674.576,A -85,B 0,C 180,E1 25924.384,E2 25924.384} C_VEL
LIN {X 0,Y 536.127,Z 682.772,A -85,B 0,C 180,E1 25922.994,E2 25922.994} C_VEL
LIN {X 0,Y 535.996,Z 690,A -85,B 0,C 180,E1 25921.39,E2 25921.39} C_VEL
LIN {X 0,Y 535.942,Z 695.492,A -85,B 0,C 180,E1 25919.787,E2 25919.787} C_VEL
LIN {X 0,Y 535.919,Z 699.626,A -85,B 0,C 180,E1 25918.076,E2 25918.076} C_VEL
LIN {X 0,Y 535.916,Z 701.746,A -85,B 0,C 180,E1 25916.471,E2 25916.471} C_VEL
LIN {X 0,Y 535.916,Z 702.406,A -85,B 0,C 180,E1 25915.064,E2 25915.064} C_VEL
LIN {X 0,Y 535.914,Z 701.87,A -85,B 0,C 180,E1 25913.573,E2 25913.573} C_VEL
LIN {X 0,Y 535.92,Z 699.428,A -85,B 0,C 180,E1 25911.741,E2 25911.741} C_VEL
LIN {X 0,Y 535.938,Z 695.774,A -85,B 0,C 180,E1 25910.226,E2 25910.226} C_VEL
LIN {X 0,Y 536.002,Z 689.984,A -85,B 0,C 180,E1 25908.487,E2 25908.487} C_VEL
LIN {X 0,Y 536.137,Z 682.458,A -85,B 0,C 180,E1 25906.849,E2 25906.849} C_VEL
LIN {X 0,Y 536.316,Z 674.782,A -85,B 0,C 180,E1 25905.534,E2 25905.534} C_VEL
LIN {X 0,Y 536.593,Z 664.36,A -85,B 0,C 180,E1 25904.103,E2 25904.103} C_VEL
LIN {X 0,Y 536.887,Z 653.112,A -85,B 0,C 180,E1 25902.888,E2 25902.888} C_VEL
LIN {X 0,Y 537.199,Z 640.381,A -85,B 0,C 180,E1 25901.779,E2 25901.779} C_VEL
LIN {X 0,Y 537.519,Z 626.479,A -85,B 0,C 180,E1 25900.834,E2 25900.834} C_VEL
LIN {X 0,Y 537.801,Z 611.508,A -85,B 0,C 180,E1 25900.053,E2 25900.053} C_VEL
LIN {X 0,Y 538.005,Z 595.789,A -85,B 0,C 180,E1 25899.465,E2 25899.465} C_VEL
LIN {X 0,Y 538.14,Z 579.443,A -85,B 0,C 180,E1 25899.065,E2 25899.065} C_VEL
LIN {X 0,Y 538.476,Z 441.471,A -85,B 0,C 180,E1 25897.18,E2 25897.18} C_VEL
LIN {X 0,Y 538.365,Z 439.639,A -85,B 0,C 180,E1 25897.1,E2 25897.1} C_VEL
LIN {X 0,Y 538.905,Z 399.026,A -85,B 0,C 180,E1 25893.896,E2 25893.896} C_VEL
LIN {X 0,Y 539.126,Z 357.684,A -85,B 0,C 180,E1 25890.746,E2 25890.746} C_VEL
LIN {X 0,Y 538.97,Z 322.553,A -85,B 0,C 180,E1 25888.174,E2 25888.174} C_VEL
LIN {X 0,Y 538.619,Z 300.685,A -85,B 0,C 180,E1 25886.653,E2 25886.653} C_VEL
LIN {X 0,Y 537.734,Z 268.453,A -85,B 0,C 180,E1 25884.53,E2 25884.53} C_VEL
LIN {X 0,Y 537.598,Z 259.868,A -85,B 0,C 180,E1 25883.972,E2 25883.972} C_VEL
LIN {X 0,Y 539.02,Z 261.262,A -85,B 0,C 180,E1 25883.72,E2 25883.72} C_VEL
LIN {X 0,Y 541.184,Z 261.343,A -85,B 0,C 180,E1 25883.494,E2 25883.494} C_VEL
LIN {X 0,Y 543.24,Z 260.818,A -85,B 0,C 180,E1 25883.327,E2 25883.327} C_VEL
LIN {X 0,Y 545.547,Z 265.044,A -85,B 0,C 180,E1 25882.785,E2 25882.785} C_VEL
LIN {X 0,Y 549.435,Z 273.062,A -85,B 0,C 180,E1 25881.828,E2 25881.828} C_VEL
LIN {X 0,Y 548.113,Z 322.603,A -85,B 0,C 180,E1 25878.464,E2 25878.464} C_VEL
LIN {X 0,Y 549.448,Z 336.589,A -85,B 0,C 180,E1 25877.395,E2 25877.395} C_VEL
LIN {X 0,Y 552.199,Z 348.337,A -85,B 0,C 180,E1 25876.38,E2 25876.38} C_VEL
LIN {X 0,Y 556.068,Z 357.517,A -85,B 0,C 180,E1 25875.473,E2 25875.473} C_VEL
LIN {X 0,Y 561.322,Z 365.349,A -85,B 0,C 180,E1 25874.573,E2 25874.573} C_VEL
LIN {X 0,Y 567.473,Z 371.414,A -85,B 0,C 180,E1 25873.748,E2 25873.748} C_VEL
LIN {X 0,Y 574.948,Z 376.264,A -85,B 0,C 180,E1 25872.935,E2 25872.935} C_VEL
LIN {X 0,Y 579.266,Z 378.039,A -85,B 0,C 180,E1 25872.447,E2 25872.447} C_VEL
LIN {X 0,Y 582.764,Z 378.541,A -85,B 0,C 180,E1 25871.868,E2 25871.868} C_VEL
LIN {X 0,Y 585.057,Z 377.712,A -85,B 0,C 180,E1 25871.24,E2 25871.24} C_VEL
LIN {X 0,Y 585.881,Z 375.746,A -85,B 0,C 180,E1 25870.616,E2 25870.616} C_VEL
LIN {X 0,Y 585.234,Z 372.782,A -85,B 0,C 180,E1 25870.034,E2 25870.034} C_VEL
LIN {X 0,Y 583.183,Z 369.066,A -85,B 0,C 180,E1 25869.532,E2 25869.532} C_VEL
LIN {X 0,Y 577.581,Z 360.924,A -85,B 0,C 180,E1 25868.821,E2 25868.821} C_VEL
LIN {X 0,Y 572.447,Z 350.953,A -85,B 0,C 180,E1 25868.177,E2 25868.177} C_VEL
LIN {X 0,Y 568.338,Z 339.717,A -85,B 0,C 180,E1 25867.647,E2 25867.647} C_VEL
LIN {X 0,Y 565.261,Z 327.32,A -85,B 0,C 180,E1 25867.241,E2 25867.241} C_VEL
LIN {X 0,Y 563.187,Z 313.498,A -85,B 0,C 180,E1 25866.963,E2 25866.963} C_VEL
LIN {X 0,Y 562.698,Z 309.409,A -85,B 0,C 180,E1 25866.897,E2 25866.897} C_VEL
LIN {X 0,Y 560.381,Z 315.962,A -85,B 0,C 180,E1 25866.58,E2 25866.58} C_VEL
LIN {X 0,Y 558.904,Z 318.818,A -85,B 0,C 180,E1 25866.375,E2 25866.375} C_VEL
LIN {X 0,Y 554.645,Z 368.036,A -85,B 0,C 180,E1 25865.774,E2 25865.774} C_VEL
LIN {X 0,Y 550.979,Z 400.28,A -85,B 0,C 180,E1 25865.241,E2 25865.241} C_VEL
LIN {X 0,Y 548.627,Z 414.407,A -85,B 0,C 180,E1 25864.892,E2 25864.892} C_VEL
LIN {X 0,Y 547.557,Z 417.729,A -85,B 0,C 180,E1 25864.731,E2 25864.731} C_VEL
LIN {X 0,Y 547.148,Z 418.318,A -85,B 0,C 180,E1 25864.665,E2 25864.665} C_VEL
LIN {X 0,Y 545.354,Z 608.526,A -85,B 0,C 180,E1 25861.826,E2 25861.826} C_VEL
LIN {X 0,Y 544.77,Z 630.508,A -85,B 0,C 180,E1 25861.305,E2 25861.305} C_VEL
LIN {X 0,Y 544.059,Z 653.317,A -85,B 0,C 180,E1 25860.541,E2 25860.541} C_VEL
LIN {X 0,Y 543.204,Z 674.555,A -85,B 0,C 180,E1 25859.619,E2 25859.619} C_VEL
LIN {X 0,Y 542.286,Z 694.785,A -85,B 0,C 180,E1 25858.525,E2 25858.525} C_VEL
LIN {X 0,Y 541.286,Z 714.98,A -85,B 0,C 180,E1 25857.206,E2 25857.206} C_VEL
LIN {X 0,Y 540.251,Z 734.823,A -85,B 0,C 180,E1 25855.663,E2 25855.663} C_VEL
LIN {X 0,Y 539.33,Z 752.83,A -85,B 0,C 180,E1 25854.012,E2 25854.012} C_VEL
LIN {X 0,Y 538.458,Z 770.22,A -85,B 0,C 180,E1 25852.145,E2 25852.145} C_VEL
LIN {X 0,Y 537.69,Z 786.413,A -85,B 0,C 180,E1 25850.105,E2 25850.105} C_VEL
LIN {X 0,Y 537.083,Z 800.888,A -85,B 0,C 180,E1 25847.955,E2 25847.955} C_VEL
LIN {X 0,Y 536.63,Z 813.27,A -85,B 0,C 180,E1 25845.785,E2 25845.785} C_VEL
LIN {X 0,Y 536.303,Z 824.315,A -85,B 0,C 180,E1 25843.476,E2 25843.476} C_VEL
LIN {X 0,Y 536.097,Z 833.329,A -85,B 0,C 180,E1 25841.18,E2 25841.18} C_VEL
LIN {X 0,Y 535.984,Z 840.396,A -85,B 0,C 180,E1 25838.907,E2 25838.907} C_VEL
LIN {X 0,Y 535.927,Z 846.009,A -85,B 0,C 180,E1 25836.535,E2 25836.535} C_VEL
LIN {X 0,Y 535.916,Z 849.738,A -85,B 0,C 180,E1 25834.28,E2 25834.28} C_VEL
LIN {X 0,Y 535.908,Z 851.9,A -85,B 0,C 180,E1 25831.925,E2 25831.925} C_VEL
LIN {X 0,Y 535.898,Z 852.442,A -85,B 0,C 180,E1 25829.572,E2 25829.572} C_VEL
LIN {X 0,Y 535.91,Z 851.331,A -85,B 0,C 180,E1 25827.219,E2 25827.219} C_VEL
LIN {X 0,Y 535.923,Z 848.486,A -85,B 0,C 180,E1 25824.862,E2 25824.862} C_VEL
LIN {X 0,Y 535.948,Z 843.936,A -85,B 0,C 180,E1 25822.496,E2 25822.496} C_VEL
LIN {X 0,Y 536.016,Z 837.924,A -85,B 0,C 180,E1 25820.227,E2 25820.227} C_VEL
LIN {X 0,Y 536.158,Z 830.096,A -85,B 0,C 180,E1 25817.944,E2 25817.944} C_VEL
LIN {X 0,Y 536.404,Z 820.353,A -85,B 0,C 180,E1 25815.646,E2 25815.646} C_VEL
LIN {X 0,Y 536.773,Z 809.12,A -85,B 0,C 180,E1 25813.441,E2 25813.441} C_VEL
LIN {X 0,Y 537.291,Z 795.627,A -85,B 0,C 180,E1 25811.219,E2 25811.219} C_VEL
LIN {X 0,Y 537.916,Z 781.191,A -85,B 0,C 180,E1 25809.205,E2 25809.205} C_VEL
LIN {X 0,Y 538.687,Z 765.207,A -85,B 0,C 180,E1 25807.29,E2 25807.29} C_VEL
LIN {X 0,Y 539.598,Z 747.528,A -85,B 0,C 180,E1 25805.476,E2 25805.476} C_VEL
LIN {X 0,Y 540.557,Z 729.316,A -85,B 0,C 180,E1 25803.881,E2 25803.881} C_VEL
LIN {X 0,Y 541.534,Z 710,A -85,B 0,C 180,E1 25802.445,E2 25802.445} C_VEL
LIN {X 0,Y 542.503,Z 689.784,A -85,B 0,C 180,E1 25801.186,E2 25801.186} C_VEL
LIN {X 0,Y 543.462,Z 668.405,A -85,B 0,C 180,E1 25800.093,E2 25800.093} C_VEL
LIN {X 0,Y 544.284,Z 646.97,A -85,B 0,C 180,E1 25799.221,E2 25799.221} C_VEL
LIN {X 0,Y 544.964,Z 624.813,A -85,B 0,C 180,E1 25798.541,E2 25798.541} C_VEL
LIN {X 0,Y 545.433,Z 602.812,A -85,B 0,C 180,E1 25798.073,E2 25798.073} C_VEL
LIN {X 0,Y 547.272,Z 417.938,A -85,B 0,C 180,E1 25795.312,E2 25795.312} C_VEL
LIN {X 0,Y 548.27,Z 415.717,A -85,B 0,C 180,E1 25795.161,E2 25795.161} C_VEL
LIN {X 0,Y 550.403,Z 404.254,A -85,B 0,C 180,E1 25794.844,E2 25794.844} C_VEL
LIN {X 0,Y 553.832,Z 376.055,A -85,B 0,C 180,E1 25794.343,E2 25794.343} C_VEL
LIN {X 0,Y 558.044,Z 329.891,A -85,B 0,C 180,E1 25793.745,E2 25793.745} C_VEL
LIN {X 0,Y 558.97,Z 319.988,A -85,B 0,C 180,E1 25793.615,E2 25793.615} C_VEL
LIN {X 0,Y 561.351,Z 315.385,A -85,B 0,C 180,E1 25793.287,E2 25793.287} C_VEL
LIN {X 0,Y 562.029,Z 313.461,A -85,B 0,C 180,E1 25793.194,E2 25793.194} C_VEL
LIN {X 0,Y 562.263,Z 339.554,A -85,B 0,C 180,E1 25793.162,E2 25793.162} C_VEL
LIN {X 0,Y 563.507,Z 354.336,A -85,B 0,C 180,E1 25792.994,E2 25792.994} C_VEL
LIN {X 0,Y 565.79,Z 367.644,A -85,B 0,C 180,E1 25792.688,E2 25792.688} C_VEL
LIN {X 0,Y 569.14,Z 379.849,A -85,B 0,C 180,E1 25792.248,E2 25792.248} C_VEL
LIN {X 0,Y 573.452,Z 390.662,A -85,B 0,C 180,E1 25791.695,E2 25791.695} C_VEL
LIN {X 0,Y 578.837,Z 400.353,A -85,B 0,C 180,E1 25791.025,E2 25791.025} C_VEL
LIN {X 0,Y 581.703,Z 405.099,A -85,B 0,C 180,E1 25790.571,E2 25790.571} C_VEL
LIN {X 0,Y 583.046,Z 408.828,A -85,B 0,C 180,E1 25790.045,E2 25790.045} C_VEL
LIN {X 0,Y 582.965,Z 411.7,A -85,B 0,C 180,E1 25789.446,E2 25789.446} C_VEL
LIN {X 0,Y 581.384,Z 413.447,A -85,B 0,C 180,E1 25788.8,E2 25788.8} C_VEL
LIN {X 0,Y 578.889,Z 413.884,A -85,B 0,C 180,E1 25788.258,E2 25788.258} C_VEL
LIN {X 0,Y 575.456,Z 413.207,A -85,B 0,C 180,E1 25787.746,E2 25787.746} C_VEL
LIN {X 0,Y 570.706,Z 410.965,A -85,B 0,C 180,E1 25787.229,E2 25787.229} C_VEL
LIN {X 0,Y 563.396,Z 405.752,A -85,B 0,C 180,E1 25786.392,E2 25786.392} C_VEL
LIN {X 0,Y 556.985,Z 398.716,A -85,B 0,C 180,E1 25785.452,E2 25785.452} C_VEL
LIN {X 0,Y 552.046,Z 390.165,A -85,B 0,C 180,E1 25784.47,E2 25784.47} C_VEL
LIN {X 0,Y 548.674,Z 380.171,A -85,B 0,C 180,E1 25783.466,E2 25783.466} C_VEL
LIN {X 0,Y 546.562,Z 367.372,A -85,B 0,C 180,E1 25782.314,E2 25782.314} C_VEL
LIN {X 0,Y 546.204,Z 351.097,A -85,B 0,C 180,E1 25780.993,E2 25780.993} C_VEL
LIN {X 0,Y 548.072,Z 309.657,A -85,B 0,C 180,E1 25777.738,E2 25777.738} C_VEL
LIN {X 0,Y 549.841,Z 274.346,A -85,B 0,C 180,E1 25774.838,E2 25774.838} C_VEL
LIN {X 0,Y 542.099,Z 258.048,A -85,B 0,C 180,E1 25772.461,E2 25772.461} C_VEL
LIN {X 0,Y 538.253,Z 250.048,A -85,B 0,C 180,E1 25771.216,E2 25771.216} C_VEL
LIN {X 0,Y 536.641,Z 246.885,A -85,B 0,C 180,E1 25770.698,E2 25770.698} C_VEL
LIN {X 0,Y 536.457,Z 245.908,A -85,B 0,C 180,E1 25770.561,E2 25770.561} C_VEL
LIN {X 0,Y 536.446,Z 246.049,A -85,B 0,C 180,E1 25767.546,E2 25767.546} C_VEL
LIN {X 0,Y 537.866,Z 251.798,A -85,B 0,C 180,E1 25767.153,E2 25767.153} C_VEL
LIN {X 0,Y 538.466,Z 295.494,A -85,B 0,C 180,E1 25764.403,E2 25764.403} C_VEL
LIN {X 0,Y 538.896,Z 335.452,A -85,B 0,C 180,E1 25761.741,E2 25761.741} C_VEL
LIN {X 0,Y 538.939,Z 370.932,A -85,B 0,C 180,E1 25759.283,E2 25759.283} C_VEL
LIN {X 0,Y 538.7,Z 412.361,A -85,B 0,C 180,E1 25756.343,E2 25756.343} C_VEL
LIN {X 0,Y 538.168,Z 456.963,A -85,B 0,C 180,E1 25753.1,E2 25753.1} C_VEL
LIN {X 0,Y 537.771,Z 489.871,A -85,B 0,C 180,E1 25750.701,E2 25750.701} C_VEL
LIN {X 0,Y 537.511,Z 603.182,A -85,B 0,C 180,E1 25749.138,E2 25749.138} C_VEL
LIN {X 0,Y 537.385,Z 617.374,A -85,B 0,C 180,E1 25748.749,E2 25748.749} C_VEL
LIN {X 0,Y 537.226,Z 631.024,A -85,B 0,C 180,E1 25748.185,E2 25748.185} C_VEL
LIN {X 0,Y 536.992,Z 644.981,A -85,B 0,C 180,E1 25747.381,E2 25747.381} C_VEL
LIN {X 0,Y 536.751,Z 658.126,A -85,B 0,C 180,E1 25746.363,E2 25746.363} C_VEL
LIN {X 0,Y 536.513,Z 669.249,A -85,B 0,C 180,E1 25745.239,E2 25745.239} C_VEL
LIN {X 0,Y 536.316,Z 679.144,A -85,B 0,C 180,E1 25743.955,E2 25743.955} C_VEL
LIN {X 0,Y 536.166,Z 686.806,A -85,B 0,C 180,E1 25742.672,E2 25742.672} C_VEL
LIN {X 0,Y 536.05,Z 693.589,A -85,B 0,C 180,E1 25741.175,E2 25741.175} C_VEL
LIN {X 0,Y 535.988,Z 698.343,A -85,B 0,C 180,E1 25739.679,E2 25739.679} C_VEL
LIN {X 0,Y 535.954,Z 701.625,A -85,B 0,C 180,E1 25738.075,E2 25738.075} C_VEL
LIN {X 0,Y 535.946,Z 702.969,A -85,B 0,C 180,E1 25736.577,E2 25736.577} C_VEL
LIN {X 0,Y 535.944,Z 702.835,A -85,B 0,C 180,E1 25735.031,E2 25735.031} C_VEL
LIN {X 0,Y 535.955,Z 700.964,A -85,B 0,C 180,E1 25733.465,E2 25733.465} C_VEL
LIN {X 0,Y 535.983,Z 697.526,A -85,B 0,C 180,E1 25731.957,E2 25731.957} C_VEL
LIN {X 0,Y 536.048,Z 692.318,A -85,B 0,C 180,E1 25730.444,E2 25730.444} C_VEL
LIN {X 0,Y 536.163,Z 685.54,A -85,B 0,C 180,E1 25729.034,E2 25729.034} C_VEL
LIN {X 0,Y 536.326,Z 676.902,A -85,B 0,C 180,E1 25727.658,E2 25727.658} C_VEL
LIN {X 0,Y 536.531,Z 666.733,A -85,B 0,C 180,E1 25726.419,E2 25726.419} C_VEL
LIN {X 0,Y 536.752,Z 655.771,A -85,B 0,C 180,E1 25725.366,E2 25725.366} C_VEL
LIN {X 0,Y 536.986,Z 643.437,A -85,B 0,C 180,E1 25724.447,E2 25724.447} C_VEL
LIN {X 0,Y 537.221,Z 629.87,A -85,B 0,C 180,E1 25723.678,E2 25723.678} C_VEL
LIN {X 0,Y 537.412,Z 614.853,A -85,B 0,C 180,E1 25723.079,E2 25723.079} C_VEL
LIN {X 0,Y 537.532,Z 600.055,A -85,B 0,C 180,E1 25722.706,E2 25722.706} C_VEL
LIN {X 0,Y 537.716,Z 489.12,A -85,B 0,C 180,E1 25721.185,E2 25721.185} C_VEL
LIN {X 0,Y 537.614,Z 487.564,A -85,B 0,C 180,E1 25721.135,E2 25721.135} C_VEL
LIN {X 0,Y 536.755,Z 481.371,A -85,B 0,C 180,E1 25720.644,E2 25720.644} C_VEL
LIN {X 0,Y 530.997,Z 465.615,A -85,B 0,C 180,E1 25719.24,E2 25719.24} C_VEL
LIN {X 0,Y 530.358,Z 460.271,A -85,B 0,C 180,E1 25718.814,E2 25718.814} C_VEL
LIN {X 0,Y 531.084,Z 413.945,A -85,B 0,C 180,E1 25715.353,E2 25715.353} C_VEL
LIN {X 0,Y 531.751,Z 369.326,A -85,B 0,C 180,E1 25712.031,E2 25712.031} C_VEL
LIN {X 0,Y 532.192,Z 326.958,A -85,B 0,C 180,E1 25708.891,E2 25708.891} C_VEL
LIN {X 0,Y 532.431,Z 285.773,A -85,B 0,C 180,E1 25705.84,E2 25705.84} C_VEL
LIN {X 0,Y 532.49,Z 260.018,A -85,B 0,C 180,E1 25703.936,E2 25703.936} C_VEL
LIN {X 0,Y 528.52,Z 246.898,A -85,B 0,C 180,E1 25702.709,E2 25702.709} C_VEL
LIN {X 0,Y 528.502,Z 246.905,A -85,B 0,C 180,E1 25699.111,E2 25699.111} C_VEL
LIN {X 0,Y 528.518,Z 246.904,A -85,B 0,C 180,E1 25695.726,E2 25695.726} C_VEL
LIN {X 0,Y 528.5,Z 246.907,A -85,B 0,C 180,E1 25692.339,E2 25692.339} C_VEL
LIN {X 0,Y 528.786,Z 248.238,A -85,B 0,C 180,E1 25692.083,E2 25692.083} C_VEL
LIN {X 0,Y 530.689,Z 252.283,A -85,B 0,C 180,E1 25691.339,E2 25691.339} C_VEL
LIN {X 0,Y 535.997,Z 264.128,A -85,B 0,C 180,E1 25689.271,E2 25689.271} C_VEL
LIN {X 0,Y 538.283,Z 270.251,A -85,B 0,C 180,E1 25688.298,E2 25688.298} C_VEL
LIN {X 0,Y 538.428,Z 272.752,A -85,B 0,C 180,E1 25687.996,E2 25687.996} C_VEL
LIN {X 0,Y 535.949,Z 304.646,A -85,B 0,C 180,E1 25684.735,E2 25684.735} C_VEL
LIN {X 0,Y 538.201,Z 315.952,A -85,B 0,C 180,E1 25684.391,E2 25684.391} C_VEL
LIN {X 0,Y 536.216,Z 524.245,A -85,B 0,C 180,E1 25681.321,E2 25681.321} C_VEL
LIN {X 0,Y 535.808,Z 562.77,A -85,B 0,C 180,E1 25680.728,E2 25680.728} C_VEL
LIN {X 0,Y 535.294,Z 583.585,A -85,B 0,C 180,E1 25680.209,E2 25680.209} C_VEL
LIN {X 0,Y 534.597,Z 603.605,A -85,B 0,C 180,E1 25679.496,E2 25679.496} C_VEL
LIN {X 0,Y 533.925,Z 621.049,A -85,B 0,C 180,E1 25678.708,E2 25678.708} C_VEL
LIN {X 0,Y 533.043,Z 640.754,A -85,B 0,C 180,E1 25677.601,E2 25677.601} C_VEL
LIN {X 0,Y 532.279,Z 656.937,A -85,B 0,C 180,E1 25676.496,E2 25676.496} C_VEL
LIN {X 0,Y 531.459,Z 673.604,A -85,B 0,C 180,E1 25675.163,E2 25675.163} C_VEL
LIN {X 0,Y 530.617,Z 689.916,A -85,B 0,C 180,E1 25673.605,E2 25673.605} C_VEL
LIN {X 0,Y 529.906,Z 704.841,A -85,B 0,C 180,E1 25671.938,E2 25671.938} C_VEL
LIN {X 0,Y 529.239,Z 719.435,A -85,B 0,C 180,E1 25669.996,E2 25669.996} C_VEL
LIN {X 0,Y 528.766,Z 731.722,A -85,B 0,C 180,E1 25668.066,E2 25668.066} C_VEL
LIN {X 0,Y 528.38,Z 742.965,A -85,B 0,C 180,E1 25665.926,E2 25665.926} C_VEL
LIN {X 0,Y 528.161,Z 751.279,A -85,B 0,C 180,E1 25664.023,E2 25664.023} C_VEL
LIN {X 0,Y 528.019,Z 759.244,A -85,B 0,C 180,E1 25661.762,E2 25661.762} C_VEL
LIN {X 0,Y 527.948,Z 764.708,A -85,B 0,C 180,E1 25659.704,E2 25659.704} C_VEL
LIN {X 0,Y 527.918,Z 768.83,A -85,B 0,C 180,E1 25657.619,E2 25657.619} C_VEL
LIN {X 0,Y 527.904,Z 771.509,A -85,B 0,C 180,E1 25655.325,E2 25655.325} C_VEL
LIN {X 0,Y 527.904,Z 772.403,A -85,B 0,C 180,E1 25653.366,E2 25653.366} C_VEL
LIN {X 0,Y 527.907,Z 771.956,A -85,B 0,C 180,E1 25651.194,E2 25651.194} C_VEL
LIN {X 0,Y 527.916,Z 769.687,A -85,B 0,C 180,E1 25648.915,E2 25648.915} C_VEL
LIN {X 0,Y 527.936,Z 766.373,A -85,B 0,C 180,E1 25646.96,E2 25646.96} C_VEL
LIN {X 0,Y 527.995,Z 760.818,A -85,B 0,C 180,E1 25644.676,E2 25644.676} C_VEL
LIN {X 0,Y 528.112,Z 753.983,A -85,B 0,C 180,E1 25642.603,E2 25642.603} C_VEL
LIN {X 0,Y 528.324,Z 745.545,A -85,B 0,C 180,E1 25640.523,E2 25640.523} C_VEL
LIN {X 0,Y 528.644,Z 735.017,A -85,B 0,C 180,E1 25638.435,E2 25638.435} C_VEL
LIN {X 0,Y 529.035,Z 724.468,A -85,B 0,C 180,E1 25636.669,E2 25636.669} C_VEL
LIN {X 0,Y 529.65,Z 710.424,A -85,B 0,C 180,E1 25634.675,E2 25634.675} C_VEL
LIN {X 0,Y 530.268,Z 696.964,A -85,B 0,C 180,E1 25633.063,E2 25633.063} C_VEL
LIN {X 0,Y 531.093,Z 680.713,A -85,B 0,C 180,E1 25631.391,E2 25631.391} C_VEL
LIN {X 0,Y 531.901,Z 664.485,A -85,B 0,C 180,E1 25629.994,E2 25629.994} C_VEL
LIN {X 0,Y 532.736,Z 647.781,A -85,B 0,C 180,E1 25628.763,E2 25628.763} C_VEL
LIN {X 0,Y 533.567,Z 629.373,A -85,B 0,C 180,E1 25627.641,E2 25627.641} C_VEL
LIN {X 0,Y 534.275,Z 612.448,A -85,B 0,C 180,E1 25626.794,E2 25626.794} C_VEL
LIN {X 0,Y 534.979,Z 593.25,A -85,B 0,C 180,E1 25626.015,E2 25626.015} C_VEL
LIN {X 0,Y 535.546,Z 573.028,A -85,B 0,C 180,E1 25625.418,E2 25625.418} C_VEL
LIN {X 0,Y 535.899,Z 555.051,A -85,B 0,C 180,E1 25625.046,E2 25625.046} C_VEL
LIN {X 0,Y 538.072,Z 329.722,A -85,B 0,C 180,E1 25621.726,E2 25621.726} C_VEL
LIN {X 0,Y 538.076,Z 311.944,A -85,B 0,C 180,E1 25621.445,E2 25621.445} C_VEL
LIN {X 0,Y 536.403,Z 302.845,A -85,B 0,C 180,E1 25621.174,E2 25621.174} C_VEL
LIN {X 0,Y 538.578,Z 270.575,A -85,B 0,C 180,E1 25618.399,E2 25618.399} C_VEL
LIN {X 0,Y 535.713,Z 262.799,A -85,B 0,C 180,E1 25617.357,E2 25617.357} C_VEL
LIN {X 0,Y 529.974,Z 250.609,A -85,B 0,C 180,E1 25615.529,E2 25615.529} C_VEL
LIN {X 0,Y 528.525,Z 246.954,A -85,B 0,C 180,E1 25615,E2 25615} C_VEL
LIN {X 0,Y 528.513,Z 246.909,A -85,B 0,C 180,E1 25611.507,E2 25611.507} C_VEL
LIN {X 0,Y 528.517,Z 246.904,A -85,B 0,C 180,E1 25608.03,E2 25608.03} C_VEL
LIN {X 0,Y 528.526,Z 246.903,A -85,B 0,C 180,E1 25604.577,E2 25604.577} C_VEL
LIN {X 0,Y 528.529,Z 246.892,A -85,B 0,C 180,E1 25600.99,E2 25600.99} C_VEL
LIN {X 0,Y 528.519,Z 246.894,A -85,B 0,C 180,E1 25597.386,E2 25597.386} C_VEL
LIN {X 0,Y 528.524,Z 246.903,A -85,B 0,C 180,E1 25593.85,E2 25593.85} C_VEL
LIN {X 0,Y 528.523,Z 246.904,A -85,B 0,C 180,E1 25590.383,E2 25590.383} C_VEL
LIN {X 0,Y 528.522,Z 246.998,A -85,B 0,C 180,E1 25588.804,E2 25588.804} C_VEL
LIN {X 0,Y 532.87,Z 261.806,A -85,B 0,C 180,E1 25587.369,E2 25587.369} C_VEL
LIN {X 0,Y 532.581,Z 305.133,A -85,B 0,C 180,E1 25583.894,E2 25583.894} C_VEL
LIN {X 0,Y 532.131,Z 345.456,A -85,B 0,C 180,E1 25580.653,E2 25580.653} C_VEL
LIN {X 0,Y 531.486,Z 387.576,A -85,B 0,C 180,E1 25577.258,E2 25577.258} C_VEL
LIN {X 0,Y 530.74,Z 429.871,A -85,B 0,C 180,E1 25573.843,E2 25573.843} C_VEL
LIN {X 0,Y 530.627,Z 440.047,A -85,B 0,C 180,E1 25573.046,E2 25573.046} C_VEL
LIN {X 0,Y 531.095,Z 447.464,A -85,B 0,C 180,E1 25572.922,E2 25572.922} C_VEL
LIN {X 0,Y 530.414,Z 582.111,A -85,B 0,C 180,E1 25571.028,E2 25571.028} C_VEL
LIN {X 0,Y 530.256,Z 598.97,A -85,B 0,C 180,E1 25570.577,E2 25570.577} C_VEL
LIN {X 0,Y 529.993,Z 614.614,A -85,B 0,C 180,E1 25569.941,E2 25569.941} C_VEL
LIN {X 0,Y 529.694,Z 629.476,A -85,B 0,C 180,E1 25569.124,E2 25569.124} C_VEL
LIN {X 0,Y 529.341,Z 643.091,A -85,B 0,C 180,E1 25568.145,E2 25568.145} C_VEL
LIN {X 0,Y 529.015,Z 655.763,A -85,B 0,C 180,E1 25567.003,E2 25567.003} C_VEL
LIN {X 0,Y 528.682,Z 667.655,A -85,B 0,C 180,E1 25565.644,E2 25565.644} C_VEL
LIN {X 0,Y 528.424,Z 677.518,A -85,B 0,C 180,E1 25564.232,E2 25564.232} C_VEL
LIN {X 0,Y 528.22,Z 686.385,A -85,B 0,C 180,E1 25562.604,E2 25562.604} C_VEL
LIN {X 0,Y 528.103,Z 693.115,A -85,B 0,C 180,E1 25560.977,E2 25560.977} C_VEL
LIN {X 0,Y 528.027,Z 698.313,A -85,B 0,C 180,E1 25559.241,E2 25559.241} C_VEL
LIN {X 0,Y 527.99,Z 701.603,A -85,B 0,C 180,E1 25557.504,E2 25557.504} C_VEL
LIN {X 0,Y 527.974,Z 703.28,A -85,B 0,C 180,E1 25555.765,E2 25555.765} C_VEL
LIN {X 0,Y 527.985,Z 703.144,A -85,B 0,C 180,E1 25553.913,E2 25553.913} C_VEL
LIN {X 0,Y 528.003,Z 701.357,A -85,B 0,C 180,E1 25552.164,E2 25552.164} C_VEL
LIN {X 0,Y 528.065,Z 697.493,A -85,B 0,C 180,E1 25550.299,E2 25550.299} C_VEL
LIN {X 0,Y 528.151,Z 692.277,A -85,B 0,C 180,E1 25548.645,E2 25548.645} C_VEL
LIN {X 0,Y 528.307,Z 684.54,A -85,B 0,C 180,E1 25546.873,E2 25546.873} C_VEL
LIN {X 0,Y 528.512,Z 676.247,A -85,B 0,C 180,E1 25545.427,E2 25545.427} C_VEL
LIN {X 0,Y 528.8,Z 665.734,A -85,B 0,C 180,E1 25543.975,E2 25543.975} C_VEL
LIN {X 0,Y 529.114,Z 654.452,A -85,B 0,C 180,E1 25542.742,E2 25542.742} C_VEL
LIN {X 0,Y 529.435,Z 641.598,A -85,B 0,C 180,E1 25541.616,E2 25541.616} C_VEL
LIN {X 0,Y 529.756,Z 627.622,A -85,B 0,C 180,E1 25540.662,E2 25540.662} C_VEL
LIN {X 0,Y 530.015,Z 613.548,A -85,B 0,C 180,E1 25539.92,E2 25539.92} C_VEL
LIN {X 0,Y 530.217,Z 598.019,A -85,B 0,C 180,E1 25539.325,E2 25539.325} C_VEL
LIN {X 0,Y 530.334,Z 581.5,A -85,B 0,C 180,E1 25538.909,E2 25538.909} C_VEL
LIN {X 0,Y 530.752,Z 442.218,A -85,B 0,C 180,E1 25536.963,E2 25536.963} C_VEL
LIN {X 0,Y 531.283,Z 401.381,A -85,B 0,C 180,E1 25533.752,E2 25533.752} C_VEL
LIN {X 0,Y 531.521,Z 360.82,A -85,B 0,C 180,E1 25530.658,E2 25530.658} C_VEL
LIN {X 0,Y 531.314,Z 320.975,A -85,B 0,C 180,E1 25527.758,E2 25527.758} C_VEL
LIN {X 0,Y 530.845,Z 297.703,A -85,B 0,C 180,E1 25526.165,E2 25526.165} C_VEL
LIN {X 0,Y 530.028,Z 267.465,A -85,B 0,C 180,E1 25524.179,E2 25524.179} C_VEL
LIN {X 0,Y 531.474,Z 268.785,A -85,B 0,C 180,E1 25523.925,E2 25523.925} C_VEL
LIN {X 0,Y 533.646,Z 268.834,A -85,B 0,C 180,E1 25523.696,E2 25523.696} C_VEL
LIN {X 0,Y 535.364,Z 268.234,A -85,B 0,C 180,E1 25523.566,E2 25523.566} C_VEL
LIN {X 0,Y 538.941,Z 268.478,A -85,B 0,C 180,E1 25523.185,E2 25523.185} C_VEL
LIN {X 0,Y 542.96,Z 277.195,A -85,B 0,C 180,E1 25522.144,E2 25522.144} C_VEL
